LIN {X 0,Y 187.073,Z 696.63,A -85,B 0,C 180,E1 -22033.993,E2 -22033.993} C_VEL
LIN {X 0,Y 186.264,Z 706.069,A -85,B 0,C 180,E1 -22036.36,E2 -22036.36} C_VEL
LIN {X 0,Y 185.581,Z 714.682,A -85,B 0,C 180,E1 -22039.085,E2 -22039.085} C_VEL
LIN {X 0,Y 185.452,Z 722.782,A -85,B 0,C 180,E1 -22042.378,E2 -22042.378} C_VEL
LIN {X 0,Y 185.879,Z 728.927,A -85,B 0,C 180,E1 -22045.663,E2 -22045.663} C_VEL
LIN {X 0,Y 186.509,Z 733.408,A -85,B 0,C 180,E1 -22048.92,E2 -22048.92} C_VEL
LIN {X 0,Y 186.681,Z 734.524,A -85,B 0,C 180,E1 -22050,E2 -22050} C_VEL
LIN {X 0,Y 185.88,Z 736.061,A -85,B 0,C 180,E1 -22052.167,E2 -22052.167} C_VEL
LIN {X 0,Y 185.102,Z 737.03,A -85,B 0,C 180,E1 -22054.355,E2 -22054.355} C_VEL
LIN {X 0,Y 184.441,Z 737.622,A -85,B 0,C 180,E1 -22057.819,E2 -22057.819} C_VEL
LIN {X 0,Y 184.416,Z 737.19,A -85,B 0,C 180,E1 -22060.984,E2 -22060.984} C_VEL
LIN {X 0,Y 184.832,Z 736.376,A -85,B 0,C 180,E1 -22063.187,E2 -22063.187} C_VEL
LIN {X 0,Y 185.593,Z 735.101,A -85,B 0,C 180,E1 -22065.371,E2 -22065.371} C_VEL
LIN {X 0,Y 187.611,Z 732.415,A -85,B 0,C 180,E1 -22068.566,E2 -22068.566} C_VEL
LIN {X 0,Y 190.356,Z 728.663,A -85,B 0,C 180,E1 -22071.666,E2 -22071.666} C_VEL
LIN {X 0,Y 193.883,Z 723.809,A -85,B 0,C 180,E1 -22074.636,E2 -22074.636} C_VEL
LIN {X 0,Y 198.128,Z 717.663,A -85,B 0,C 180,E1 -22077.46,E2 -22077.46} C_VEL
LIN {X 0,Y 203.13,Z 709.985,A -85,B 0,C 180,E1 -22080.11,E2 -22080.11} C_VEL
LIN {X 0,Y 208.674,Z 700.543,A -85,B 0,C 180,E1 -22082.606,E2 -22082.606} C_VEL
LIN {X 0,Y 213.814,Z 690.855,A -85,B 0,C 180,E1 -22084.54,E2 -22084.54} C_VEL
LIN {X 0,Y 218.839,Z 680.033,A -85,B 0,C 180,E1 -22086.164,E2 -22086.164} C_VEL
LIN {X 0,Y 223.644,Z 667.781,A -85,B 0,C 180,E1 -22087.568,E2 -22087.568} C_VEL
LIN {X 0,Y 227.072,Z 655.896,A -85,B 0,C 180,E1 -22088.76,E2 -22088.76} C_VEL
LIN {X 0,Y 229.32,Z 643.699,A -85,B 0,C 180,E1 -22089.904,E2 -22089.904} C_VEL
LIN {X 0,Y 230.194,Z 631.94,A -85,B 0,C 180,E1 -22091.105,E2 -22091.105} C_VEL
LIN {X 0,Y 230.347,Z 618.408,A -85,B 0,C 180,E1 -22092.713,E2 -22092.713} C_VEL
LIN {X 0,Y 230.219,Z 613.273,A -85,B 0,C 180,E1 -22093.463,E2 -22093.463} C_VEL
LIN {X 0,Y 228.941,Z 606.861,A -85,B 0,C 180,E1 -22095.34,E2 -22095.34} C_VEL
LIN {X 0,Y 227.692,Z 600.839,A -85,B 0,C 180,E1 -22097.501,E2 -22097.501} C_VEL
LIN {X 0,Y 227.171,Z 599.159,A -85,B 0,C 180,E1 -22098.473,E2 -22098.473} C_VEL
LIN {X 0,Y 225.431,Z 596.58,A -85,B 0,C 180,E1 -22101.958,E2 -22101.958} C_VEL
LIN {X 0,Y 225.098,Z 595.189,A -85,B 0,C 180,E1 -22103.615,E2 -22103.615} C_VEL
LIN {X 0,Y 224.948,Z 594.902,A -85,B 0,C 180,E1 -22105.781,E2 -22105.781} C_VEL
LIN {X 0,Y 225.214,Z 595.291,A -85,B 0,C 180,E1 -22107.961,E2 -22107.961} C_VEL
LIN {X 0,Y 226.659,Z 598.492,A -85,B 0,C 180,E1 -22111.962,E2 -22111.962} C_VEL
LIN {X 0,Y 227.457,Z 599.455,A -85,B 0,C 180,E1 -22113.163,E2 -22113.163} C_VEL
LIN {X 0,Y 229.844,Z 603.626,A -85,B 0,C 180,E1 -22116.036,E2 -22116.036} C_VEL
LIN {X 0,Y 232.174,Z 607.948,A -85,B 0,C 180,E1 -22118.251,E2 -22118.251} C_VEL
LIN {X 0,Y 234.9,Z 614.48,A -85,B 0,C 180,E1 -22120.836,E2 -22120.836} C_VEL
LIN {X 0,Y 235.052,Z 614.986,A -85,B 0,C 180,E1 -22121,E2 -22121} C_VEL
LIN {X 0,Y 232.571,Z 626.818,A -85,B 0,C 180,E1 -22122.138,E2 -22122.138} C_VEL
LIN {X 0,Y 229.272,Z 638.439,A -85,B 0,C 180,E1 -22123.564,E2 -22123.564} C_VEL
LIN {X 0,Y 225.173,Z 649.567,A -85,B 0,C 180,E1 -22125.36,E2 -22125.36} C_VEL
LIN {X 0,Y 221.221,Z 658.24,A -85,B 0,C 180,E1 -22127.152,E2 -22127.152} C_VEL
LIN {X 0,Y 216.836,Z 666.323,A -85,B 0,C 180,E1 -22129.26,E2 -22129.26} C_VEL
LIN {X 0,Y 212.196,Z 673.689,A -85,B 0,C 180,E1 -22131.705,E2 -22131.705} C_VEL
LIN {X 0,Y 207.957,Z 679.351,A -85,B 0,C 180,E1 -22134.182,E2 -22134.182} C_VEL
LIN {X 0,Y 204.161,Z 683.648,A -85,B 0,C 180,E1 -22136.624,E2 -22136.624} C_VEL
LIN {X 0,Y 199.63,Z 687.906,A -85,B 0,C 180,E1 -22140.001,E2 -22140.001} C_VEL
LIN {X 0,Y 196.952,Z 689.883,A -85,B 0,C 180,E1 -22142.402,E2 -22142.402} C_VEL
LIN {X 0,Y 195.179,Z 690.897,A -85,B 0,C 180,E1 -22144.131,E2 -22144.131} C_VEL
LIN {X 0,Y 193.199,Z 691.679,A -85,B 0,C 180,E1 -22146.266,E2 -22146.266} C_VEL
LIN {X 0,Y 191.455,Z 691.968,A -85,B 0,C 180,E1 -22148.444,E2 -22148.444} C_VEL
LIN {X 0,Y 189.965,Z 691.804,A -85,B 0,C 180,E1 -22150.661,E2 -22150.661} C_VEL
LIN {X 0,Y 188.205,Z 690.717,A -85,B 0,C 180,E1 -22153.863,E2 -22153.863} C_VEL
LIN {X 0,Y 186.809,Z 688.3,A -85,B 0,C 180,E1 -22157.517,E2 -22157.517} C_VEL
LIN {X 0,Y 186.045,Z 684.811,A -85,B 0,C 180,E1 -22161.032,E2 -22161.032} C_VEL
LIN {X 0,Y 185.795,Z 679.7,A -85,B 0,C 180,E1 -22164.795,E2 -22164.795} C_VEL
LIN {X 0,Y 186.113,Z 673.685,A -85,B 0,C 180,E1 -22168.167,E2 -22168.167} C_VEL
LIN {X 0,Y 186.657,Z 666.806,A -85,B 0,C 180,E1 -22171.257,E2 -22171.257} C_VEL
LIN {X 0,Y 187.547,Z 658.71,A -85,B 0,C 180,E1 -22174.202,E2 -22174.202} C_VEL
LIN {X 0,Y 188.726,Z 648.29,A -85,B 0,C 180,E1 -22177.24,E2 -22177.24} C_VEL
LIN {X 0,Y 189.888,Z 637.77,A -85,B 0,C 180,E1 -22179.677,E2 -22179.677} C_VEL
LIN {X 0,Y 191.08,Z 626.638,A -85,B 0,C 180,E1 -22181.739,E2 -22181.739} C_VEL
LIN {X 0,Y 192.124,Z 614.599,A -85,B 0,C 180,E1 -22183.476,E2 -22183.476} C_VEL
LIN {X 0,Y 193.024,Z 600.995,A -85,B 0,C 180,E1 -22184.933,E2 -22184.933} C_VEL
LIN {X 0,Y 193.538,Z 586.899,A -85,B 0,C 180,E1 -22185.94,E2 -22185.94} C_VEL
LIN {X 0,Y 193.468,Z 578.507,A -85,B 0,C 180,E1 -22186.408,E2 -22186.408} C_VEL
LIN {X 0,Y 185.856,Z 553.298,A -85,B 0,C 180,E1 -22188.311,E2 -22188.311} C_VEL
LIN {X 0,Y 185.644,Z 552.294,A -85,B 0,C 180,E1 -22188.703,E2 -22188.703} C_VEL
LIN {X 0,Y 185.561,Z 552.183,A -85,B 0,C 180,E1 -22192.701,E2 -22192.701} C_VEL
LIN {X 0,Y 185.547,Z 552.185,A -85,B 0,C 180,E1 -22197.977,E2 -22197.977} C_VEL
LIN {X 0,Y 185.584,Z 552.179,A -85,B 0,C 180,E1 -22200.577,E2 -22200.577} C_VEL
LIN {X 0,Y 185.591,Z 552.18,A -85,B 0,C 180,E1 -22205.384,E2 -22205.384} C_VEL
LIN {X 0,Y 185.676,Z 552.168,A -85,B 0,C 180,E1 -22211.136,E2 -22211.136} C_VEL
LIN {X 0,Y 185.686,Z 552.163,A -85,B 0,C 180,E1 -22214.637,E2 -22214.637} C_VEL
LIN {X 0,Y 185.892,Z 552.142,A -85,B 0,C 180,E1 -22219.419,E2 -22219.419} C_VEL
LIN {X 0,Y 185.945,Z 552.131,A -85,B 0,C 180,E1 -22223.49,E2 -22223.49} C_VEL
LIN {X 0,Y 186.209,Z 552.103,A -85,B 0,C 180,E1 -22227.837,E2 -22227.837} C_VEL
LIN {X 0,Y 186.411,Z 552.074,A -85,B 0,C 180,E1 -22230,E2 -22230} C_VEL
LIN {X 0,Y 185.918,Z 552.138,A -85,B 0,C 180,E1 -22234.336,E2 -22234.336} C_VEL
LIN {X 0,Y 185.983,Z 552.127,A -85,B 0,C 180,E1 -22238.694,E2 -22238.694} C_VEL
LIN {X 0,Y 185.734,Z 552.159,A -85,B 0,C 180,E1 -22243.122,E2 -22243.122} C_VEL
LIN {X 0,Y 185.694,Z 552.166,A -85,B 0,C 180,E1 -22247.624,E2 -22247.624} C_VEL
LIN {X 0,Y 185.585,Z 552.18,A -85,B 0,C 180,E1 -22252.252,E2 -22252.252} C_VEL
LIN {X 0,Y 185.561,Z 552.178,A -85,B 0,C 180,E1 -22257.032,E2 -22257.032} C_VEL
LIN {X 0,Y 185.58,Z 552.177,A -85,B 0,C 180,E1 -22259.492,E2 -22259.492} C_VEL
LIN {X 0,Y 185.522,Z 552.185,A -85,B 0,C 180,E1 -22264.626,E2 -22264.626} C_VEL
LIN {X 0,Y 185.57,Z 552.175,A -85,B 0,C 180,E1 -22267.313,E2 -22267.313} C_VEL
LIN {X 0,Y 185.563,Z 552.182,A -85,B 0,C 180,E1 -22270.756,E2 -22270.756} C_VEL
LIN {X 0,Y 185.555,Z 552.183,A -85,B 0,C 180,E1 -22273.974,E2 -22273.974} C_VEL
LIN {X 0,Y 185.493,Z 552.19,A -85,B 0,C 180,E1 -22279.266,E2 -22279.266} C_VEL
LIN {X 0,Y 185.544,Z 552.182,A -85,B 0,C 180,E1 -22282.695,E2 -22282.695} C_VEL
LIN {X 0,Y 185.544,Z 552.185,A -85,B 0,C 180,E1 -22287.974,E2 -22287.974} C_VEL
LIN {X 0,Y 185.581,Z 552.18,A -85,B 0,C 180,E1 -22290.575,E2 -22290.575} C_VEL
LIN {X 0,Y 185.605,Z 552.174,A -85,B 0,C 180,E1 -22295.384,E2 -22295.384} C_VEL
LIN {X 0,Y 185.708,Z 552.161,A -85,B 0,C 180,E1 -22301.101,E2 -22301.101} C_VEL
LIN {X 0,Y 185.731,Z 552.161,A -85,B 0,C 180,E1 -22306.876,E2 -22306.876} C_VEL
LIN {X 0,Y 186.011,Z 552.12,A -85,B 0,C 180,E1 -22311.307,E2 -22311.307} C_VEL
LIN {X 0,Y 186.205,Z 552.101,A -85,B 0,C 180,E1 -22317.836,E2 -22317.836} C_VEL
LIN {X 0,Y 186.403,Z 552.074,A -85,B 0,C 180,E1 -22319.999,E2 -22319.999} C_VEL
LIN {X 0,Y 185.92,Z 552.139,A -85,B 0,C 180,E1 -22324.335,E2 -22324.335} C_VEL
LIN {X 0,Y 186.005,Z 552.124,A -85,B 0,C 180,E1 -22328.692,E2 -22328.692} C_VEL
LIN {X 0,Y 185.76,Z 552.158,A -85,B 0,C 180,E1 -22333.12,E2 -22333.12} C_VEL
LIN {X 0,Y 185.67,Z 552.167,A -85,B 0,C 180,E1 -22338.865,E2 -22338.865} C_VEL
LIN {X 0,Y 185.574,Z 552.181,A -85,B 0,C 180,E1 -22344.646,E2 -22344.646} C_VEL
LIN {X 0,Y 185.576,Z 552.179,A -85,B 0,C 180,E1 -22349.493,E2 -22349.493} C_VEL
LIN {X 0,Y 185.496,Z 552.189,A -85,B 0,C 180,E1 -22354.632,E2 -22354.632} C_VEL
LIN {X 0,Y 185.502,Z 552.188,A -85,B 0,C 180,E1 -22357.313,E2 -22357.313} C_VEL
LIN {X 0,Y 185.468,Z 552.196,A -85,B 0,C 180,E1 -22360.725,E2 -22360.725} C_VEL
LIN {X 0,Y 185.481,Z 552.192,A -85,B 0,C 180,E1 -22366.047,E2 -22366.047} C_VEL
LIN {X 0,Y 185.546,Z 552.184,A -85,B 0,C 180,E1 -22369.917,E2 -22369.917} C_VEL
LIN {X 0,Y 185.936,Z 552.249,A -85,B 0,C 180,E1 -22373.802,E2 -22373.802} C_VEL
LIN {X 0,Y 188.152,Z 562.25,A -85,B 0,C 180,E1 -22379.216,E2 -22379.216} C_VEL
LIN {X 0,Y 187.814,Z 565.476,A -85,B 0,C 180,E1 -22380.892,E2 -22380.892} C_VEL
LIN {X 0,Y 187.128,Z 569.009,A -85,B 0,C 180,E1 -22382.609,E2 -22382.609} C_VEL
LIN {X 0,Y 187.031,Z 577.205,A -85,B 0,C 180,E1 -22383.198,E2 -22383.198} C_VEL
LIN {X 0,Y 188.442,Z 619.399,A -85,B 0,C 180,E1 -22385.888,E2 -22385.888} C_VEL
LIN {X 0,Y 190.503,Z 655.952,A -85,B 0,C 180,E1 -22388.293,E2 -22388.293} C_VEL
LIN {X 0,Y 189.725,Z 669.284,A -85,B 0,C 180,E1 -22389.538,E2 -22389.538} C_VEL
LIN {X 0,Y 188.888,Z 680.435,A -85,B 0,C 180,E1 -22391.001,E2 -22391.001} C_VEL
LIN {X 0,Y 187.691,Z 691.166,A -85,B 0,C 180,E1 -22392.85,E2 -22392.85} C_VEL
LIN {X 0,Y 187.073,Z 696.63,A -85,B 0,C 180,E1 -22393.993,E2 -22393.993} C_VEL
LIN {X 0,Y 186.033,Z 701.223,A -85,B 0,C 180,E1 -22395.088,E2 -22395.088} C_VEL
LIN {X 0,Y 184.084,Z 705.387,A -85,B 0,C 180,E1 -22396.259,E2 -22396.259} C_VEL
LIN {X 0,Y 179.28,Z 714.053,A -85,B 0,C 180,E1 -22399.363,E2 -22399.363} C_VEL
LIN {X 0,Y 178.5,Z 717.649,A -85,B 0,C 180,E1 -22400.862,E2 -22400.862} C_VEL
LIN {X 0,Y 178.611,Z 723.876,A -85,B 0,C 180,E1 -22403.788,E2 -22403.788} C_VEL
LIN {X 0,Y 179.114,Z 728.664,A -85,B 0,C 180,E1 -22406.626,E2 -22406.626} C_VEL
LIN {X 0,Y 179.742,Z 732.818,A -85,B 0,C 180,E1 -22410,E2 -22410} C_VEL
LIN {X 0,Y 178.911,Z 734.455,A -85,B 0,C 180,E1 -22412.251,E2 -22412.251} C_VEL
LIN {X 0,Y 178.117,Z 735.55,A -85,B 0,C 180,E1 -22414.526,E2 -22414.526} C_VEL
LIN {X 0,Y 177.451,Z 736.328,A -85,B 0,C 180,E1 -22418.061,E2 -22418.061} C_VEL
LIN {X 0,Y 177.457,Z 736.091,A -85,B 0,C 180,E1 -22421.421,E2 -22421.421} C_VEL
LIN {X 0,Y 177.911,Z 735.399,A -85,B 0,C 180,E1 -22423.71,E2 -22423.71} C_VEL
LIN {X 0,Y 178.744,Z 734.306,A -85,B 0,C 180,E1 -22425.975,E2 -22425.975} C_VEL
LIN {X 0,Y 180.087,Z 732.766,A -85,B 0,C 180,E1 -22428.192,E2 -22428.192} C_VEL
LIN {X 0,Y 182.694,Z 729.638,A -85,B 0,C 180,E1 -22431.435,E2 -22431.435} C_VEL
LIN {X 0,Y 186.137,Z 725.46,A -85,B 0,C 180,E1 -22434.539,E2 -22434.539} C_VEL
LIN {X 0,Y 190.307,Z 720.092,A -85,B 0,C 180,E1 -22437.491,E2 -22437.491} C_VEL
LIN {X 0,Y 195.237,Z 713.418,A -85,B 0,C 180,E1 -22440.261,E2 -22440.261} C_VEL
LIN {X 0,Y 200.824,Z 705.139,A -85,B 0,C 180,E1 -22442.848,E2 -22442.848} C_VEL
LIN {X 0,Y 205.901,Z 696.719,A -85,B 0,C 180,E1 -22444.87,E2 -22444.87} C_VEL
LIN {X 0,Y 211.445,Z 686.511,A -85,B 0,C 180,E1 -22446.746,E2 -22446.746} C_VEL
LIN {X 0,Y 216.807,Z 675.161,A -85,B 0,C 180,E1 -22448.311,E2 -22448.311} C_VEL
LIN {X 0,Y 221.508,Z 662.765,A -85,B 0,C 180,E1 -22449.655,E2 -22449.655} C_VEL
LIN {X 0,Y 225.007,Z 649.325,A -85,B 0,C 180,E1 -22450.989,E2 -22450.989} C_VEL
LIN {X 0,Y 226.845,Z 637.084,A -85,B 0,C 180,E1 -22452.264,E2 -22452.264} C_VEL
LIN {X 0,Y 227.432,Z 624.858,A -85,B 0,C 180,E1 -22453.702,E2 -22453.702} C_VEL
LIN {X 0,Y 227.525,Z 617.57,A -85,B 0,C 180,E1 -22454.73,E2 -22454.73} C_VEL
LIN {X 0,Y 226.586,Z 612.063,A -85,B 0,C 180,E1 -22456.419,E2 -22456.419} C_VEL
LIN {X 0,Y 225.732,Z 606.668,A -85,B 0,C 180,E1 -22458.405,E2 -22458.405} C_VEL
LIN {X 0,Y 225.345,Z 605.805,A -85,B 0,C 180,E1 -22459.086,E2 -22459.086} C_VEL
LIN {X 0,Y 223.72,Z 602.433,A -85,B 0,C 180,E1 -22463.455,E2 -22463.455} C_VEL
LIN {X 0,Y 223.648,Z 601.921,A -85,B 0,C 180,E1 -22464.787,E2 -22464.787} C_VEL
LIN {X 0,Y 223.817,Z 602.217,A -85,B 0,C 180,E1 -22467.737,E2 -22467.737} C_VEL
LIN {X 0,Y 225.184,Z 605.393,A -85,B 0,C 180,E1 -22471.762,E2 -22471.762} C_VEL
LIN {X 0,Y 225.852,Z 606.361,A -85,B 0,C 180,E1 -22472.877,E2 -22472.877} C_VEL
LIN {X 0,Y 227.992,Z 610.487,A -85,B 0,C 180,E1 -22475.714,E2 -22475.714} C_VEL
LIN {X 0,Y 229.929,Z 614.71,A -85,B 0,C 180,E1 -22477.925,E2 -22477.925} C_VEL
LIN {X 0,Y 231.347,Z 619.083,A -85,B 0,C 180,E1 -22479.72,E2 -22479.72} C_VEL
LIN {X 0,Y 228.581,Z 630.79,A -85,B 0,C 180,E1 -22480.905,E2 -22480.905} C_VEL
LIN {X 0,Y 225.152,Z 641.388,A -85,B 0,C 180,E1 -22482.282,E2 -22482.282} C_VEL
LIN {X 0,Y 221.407,Z 650.703,A -85,B 0,C 180,E1 -22483.815,E2 -22483.815} C_VEL
LIN {X 0,Y 217.257,Z 659.441,A -85,B 0,C 180,E1 -22485.613,E2 -22485.613} C_VEL
LIN {X 0,Y 212.83,Z 667.182,A -85,B 0,C 180,E1 -22487.606,E2 -22487.606} C_VEL
LIN {X 0,Y 207.533,Z 675.048,A -85,B 0,C 180,E1 -22490.252,E2 -22490.252} C_VEL
LIN {X 0,Y 202.496,Z 681.229,A -85,B 0,C 180,E1 -22493.024,E2 -22493.024} C_VEL
LIN {X 0,Y 197.859,Z 686.015,A -85,B 0,C 180,E1 -22495.927,E2 -22495.927} C_VEL
LIN {X 0,Y 195.01,Z 688.451,A -85,B 0,C 180,E1 -22497.935,E2 -22497.935} C_VEL
LIN {X 0,Y 192.388,Z 690.37,A -85,B 0,C 180,E1 -22500.001,E2 -22500.001} C_VEL
LIN {X 0,Y 189.895,Z 691.813,A -85,B 0,C 180,E1 -22502.229,E2 -22502.229} C_VEL
LIN {X 0,Y 187.822,Z 692.692,A -85,B 0,C 180,E1 -22504.293,E2 -22504.293} C_VEL
LIN {X 0,Y 184.566,Z 693.194,A -85,B 0,C 180,E1 -22508.105,E2 -22508.105} C_VEL
LIN {X 0,Y 182.57,Z 692.633,A -85,B 0,C 180,E1 -22511.098,E2 -22511.098} C_VEL
LIN {X 0,Y 181.043,Z 691.349,A -85,B 0,C 180,E1 -22513.961,E2 -22513.961} C_VEL
LIN {X 0,Y 179.879,Z 689.194,A -85,B 0,C 180,E1 -22517.04,E2 -22517.04} C_VEL
LIN {X 0,Y 179.007,Z 685.579,A -85,B 0,C 180,E1 -22520.693,E2 -22520.693} C_VEL
LIN {X 0,Y 178.724,Z 680.904,A -85,B 0,C 180,E1 -22524.205,E2 -22524.205} C_VEL
LIN {X 0,Y 178.998,Z 674.136,A -85,B 0,C 180,E1 -22528.11,E2 -22528.11} C_VEL
LIN {X 0,Y 179.537,Z 667.323,A -85,B 0,C 180,E1 -22531.244,E2 -22531.244} C_VEL
LIN {X 0,Y 180.491,Z 658.88,A -85,B 0,C 180,E1 -22534.376,E2 -22534.376} C_VEL
LIN {X 0,Y 181.534,Z 649.389,A -85,B 0,C 180,E1 -22537.224,E2 -22537.224} C_VEL
LIN {X 0,Y 182.757,Z 638.966,A -85,B 0,C 180,E1 -22539.728,E2 -22539.728} C_VEL
LIN {X 0,Y 183.988,Z 627.382,A -85,B 0,C 180,E1 -22541.95,E2 -22541.95} C_VEL
LIN {X 0,Y 185.129,Z 614.5,A -85,B 0,C 180,E1 -22543.84,E2 -22543.84} C_VEL
LIN {X 0,Y 185.988,Z 602.146,A -85,B 0,C 180,E1 -22545.191,E2 -22545.191} C_VEL
LIN {X 0,Y 186.568,Z 587.713,A -85,B 0,C 180,E1 -22546.257,E2 -22546.257} C_VEL
LIN {X 0,Y 186.617,Z 580.167,A -85,B 0,C 180,E1 -22546.69,E2 -22546.69} C_VEL
LIN {X 0,Y 178.719,Z 553.941,A -85,B 0,C 180,E1 -22548.778,E2 -22548.778} C_VEL
LIN {X 0,Y 178.543,Z 553.135,A -85,B 0,C 180,E1 -22549.203,E2 -22549.203} C_VEL
LIN {X 0,Y 178.46,Z 553.068,A -85,B 0,C 180,E1 -22553.793,E2 -22553.793} C_VEL
LIN {X 0,Y 178.493,Z 553.063,A -85,B 0,C 180,E1 -22556.549,E2 -22556.549} C_VEL
LIN {X 0,Y 178.525,Z 553.059,A -85,B 0,C 180,E1 -22560.007,E2 -22560.007} C_VEL
LIN {X 0,Y 178.537,Z 553.057,A -85,B 0,C 180,E1 -22564.877,E2 -22564.877} C_VEL
LIN {X 0,Y 178.624,Z 553.045,A -85,B 0,C 180,E1 -22570.787,E2 -22570.787} C_VEL
LIN {X 0,Y 178.654,Z 553.042,A -85,B 0,C 180,E1 -22576.348,E2 -22576.348} C_VEL
LIN {X 0,Y 178.912,Z 553.008,A -85,B 0,C 180,E1 -22580.96,E2 -22580.96} C_VEL
LIN {X 0,Y 179.154,Z 552.982,A -85,B 0,C 180,E1 -22587.752,E2 -22587.752} C_VEL
LIN {X 0,Y 179.374,Z 552.95,A -85,B 0,C 180,E1 -22590,E2 -22590} C_VEL
LIN {X 0,Y 178.866,Z 553.016,A -85,B 0,C 180,E1 -22594.507,E2 -22594.507} C_VEL
LIN {X 0,Y 178.912,Z 553.007,A -85,B 0,C 180,E1 -22599.04,E2 -22599.04} C_VEL
LIN {X 0,Y 178.662,Z 553.042,A -85,B 0,C 180,E1 -22603.652,E2 -22603.652} C_VEL
LIN {X 0,Y 178.626,Z 553.041,A -85,B 0,C 180,E1 -22609.215,E2 -22609.215} C_VEL
LIN {X 0,Y 178.523,Z 553.058,A -85,B 0,C 180,E1 -22615.113,E2 -22615.113} C_VEL
LIN {X 0,Y 178.524,Z 553.058,A -85,B 0,C 180,E1 -22619.992,E2 -22619.992} C_VEL
LIN {X 0,Y 178.486,Z 553.063,A -85,B 0,C 180,E1 -22624.218,E2 -22624.218} C_VEL
LIN {X 0,Y 178.474,Z 553.063,A -85,B 0,C 180,E1 -22629.053,E2 -22629.053} C_VEL
LIN {X 0,Y 178.499,Z 553.064,A -85,B 0,C 180,E1 -22632.015,E2 -22632.015} C_VEL
LIN {X 0,Y 178.457,Z 553.063,A -85,B 0,C 180,E1 -22635.143,E2 -22635.143} C_VEL
LIN {X 0,Y 178.424,Z 553.072,A -85,B 0,C 180,E1 -22638.45,E2 -22638.45} C_VEL
LIN {X 0,Y 178.449,Z 553.066,A -85,B 0,C 180,E1 -22643.788,E2 -22643.788} C_VEL
LIN {X 0,Y 178.49,Z 553.063,A -85,B 0,C 180,E1 -22646.546,E2 -22646.546} C_VEL
LIN {X 0,Y 178.522,Z 553.061,A -85,B 0,C 180,E1 -22650.005,E2 -22650.005} C_VEL
LIN {X 0,Y 178.534,Z 553.055,A -85,B 0,C 180,E1 -22654.874,E2 -22654.874} C_VEL
LIN {X 0,Y 178.651,Z 553.04,A -85,B 0,C 180,E1 -22660.755,E2 -22660.755} C_VEL
LIN {X 0,Y 178.659,Z 553.044,A -85,B 0,C 180,E1 -22666.347,E2 -22666.347} C_VEL
LIN {X 0,Y 178.961,Z 552.999,A -85,B 0,C 180,E1 -22670.961,E2 -22670.961} C_VEL
LIN {X 0,Y 179.151,Z 552.98,A -85,B 0,C 180,E1 -22677.751,E2 -22677.751} C_VEL
LIN {X 0,Y 179.366,Z 552.951,A -85,B 0,C 180,E1 -22679.999,E2 -22679.999} C_VEL
LIN {X 0,Y 178.869,Z 553.018,A -85,B 0,C 180,E1 -22684.506,E2 -22684.506} C_VEL
LIN {X 0,Y 178.934,Z 553.003,A -85,B 0,C 180,E1 -22689.038,E2 -22689.038} C_VEL
LIN {X 0,Y 178.677,Z 553.039,A -85,B 0,C 180,E1 -22693.65,E2 -22693.65} C_VEL
LIN {X 0,Y 178.617,Z 553.045,A -85,B 0,C 180,E1 -22699.213,E2 -22699.213} C_VEL
LIN {X 0,Y 178.516,Z 553.058,A -85,B 0,C 180,E1 -22705.114,E2 -22705.114} C_VEL
LIN {X 0,Y 178.498,Z 553.064,A -85,B 0,C 180,E1 -22710.786,E2 -22710.786} C_VEL
LIN {X 0,Y 178.482,Z 553.063,A -85,B 0,C 180,E1 -22714.219,E2 -22714.219} C_VEL
LIN {X 0,Y 178.392,Z 553.076,A -85,B 0,C 180,E1 -22719.074,E2 -22719.074} C_VEL
LIN {X 0,Y 178.396,Z 553.074,A -85,B 0,C 180,E1 -22722.045,E2 -22722.045} C_VEL
LIN {X 0,Y 178.401,Z 553.075,A -85,B 0,C 180,E1 -22725.161,E2 -22725.161} C_VEL
LIN {X 0,Y 178.532,Z 553.06,A -85,B 0,C 180,E1 -22730.962,E2 -22730.962} C_VEL
LIN {X 0,Y 178.947,Z 553.155,A -85,B 0,C 180,E1 -22734.096,E2 -22734.096} C_VEL
LIN {X 0,Y 180.808,Z 561.446,A -85,B 0,C 180,E1 -22738.774,E2 -22738.774} C_VEL
LIN {X 0,Y 180.938,Z 564.291,A -85,B 0,C 180,E1 -22740.315,E2 -22740.315} C_VEL
LIN {X 0,Y 180.257,Z 567.596,A -85,B 0,C 180,E1 -22742.026,E2 -22742.026} C_VEL
LIN {X 0,Y 180.117,Z 573.051,A -85,B 0,C 180,E1 -22742.48,E2 -22742.48} C_VEL
LIN {X 0,Y 180.81,Z 605.623,A -85,B 0,C 180,E1 -22744.652,E2 -22744.652} C_VEL
LIN {X 0,Y 183.445,Z 655.478,A -85,B 0,C 180,E1 -22748.067,E2 -22748.067} C_VEL
LIN {X 0,Y 182.729,Z 668.104,A -85,B 0,C 180,E1 -22749.307,E2 -22749.307} C_VEL
LIN {X 0,Y 181.897,Z 679.224,A -85,B 0,C 180,E1 -22750.828,E2 -22750.828} C_VEL
LIN {X 0,Y 180.706,Z 689.958,A -85,B 0,C 180,E1 -22752.75,E2 -22752.75} C_VEL
LIN {X 0,Y 179.625,Z 699.71,A -85,B 0,C 180,E1 -22754.977,E2 -22754.977} C_VEL
LIN {X 0,Y 178.966,Z 708.573,A -85,B 0,C 180,E1 -22757.527,E2 -22757.527} C_VEL
LIN {X 0,Y 178.513,Z 716.871,A -85,B 0,C 180,E1 -22760.532,E2 -22760.532} C_VEL
LIN {X 0,Y 178.5,Z 717.649,A -85,B 0,C 180,E1 -22760.862,E2 -22760.862} C_VEL
LIN {X 0,Y 178.053,Z 721.046,A -85,B 0,C 180,E1 -22762.422,E2 -22762.422} C_VEL
LIN {X 0,Y 177.018,Z 724.021,A -85,B 0,C 180,E1 -22764.053,E2 -22764.053} C_VEL
LIN {X 0,Y 176.142,Z 725.771,A -85,B 0,C 180,E1 -22765.176,E2 -22765.176} C_VEL
LIN {X 0,Y 173.45,Z 729.979,A -85,B 0,C 180,E1 -22768.766,E2 -22768.766} C_VEL
LIN {X 0,Y 172.796,Z 731.035,A -85,B 0,C 180,E1 -22770.029,E2 -22770.029} C_VEL
LIN {X 0,Y 171.96,Z 732.784,A -85,B 0,C 180,E1 -22772.342,E2 -22772.342} C_VEL
LIN {X 0,Y 171.16,Z 734.013,A -85,B 0,C 180,E1 -22774.71,E2 -22774.71} C_VEL
LIN {X 0,Y 170.456,Z 734.967,A -85,B 0,C 180,E1 -22778.302,E2 -22778.302} C_VEL
LIN {X 0,Y 170.516,Z 734.937,A -85,B 0,C 180,E1 -22781.892,E2 -22781.892} C_VEL
LIN {X 0,Y 171.014,Z 734.404,A -85,B 0,C 180,E1 -22784.274,E2 -22784.274} C_VEL
LIN {X 0,Y 171.924,Z 733.425,A -85,B 0,C 180,E1 -22786.627,E2 -22786.627} C_VEL
LIN {X 0,Y 173.339,Z 732.075,A -85,B 0,C 180,E1 -22788.926,E2 -22788.926} C_VEL
LIN {X 0,Y 176.103,Z 729.219,A -85,B 0,C 180,E1 -22792.279,E2 -22792.279} C_VEL
LIN {X 0,Y 179.696,Z 725.321,A -85,B 0,C 180,E1 -22795.48,E2 -22795.48} C_VEL
LIN {X 0,Y 184.057,Z 720.321,A -85,B 0,C 180,E1 -22798.508,E2 -22798.508} C_VEL
LIN {X 0,Y 190.101,Z 712.857,A -85,B 0,C 180,E1 -22801.79,E2 -22801.79} C_VEL
LIN {X 0,Y 195.944,Z 704.787,A -85,B 0,C 180,E1 -22804.395,E2 -22804.395} C_VEL
LIN {X 0,Y 201.286,Z 696.68,A -85,B 0,C 180,E1 -22806.409,E2 -22806.409} C_VEL
LIN {X 0,Y 207.059,Z 686.823,A -85,B 0,C 180,E1 -22808.274,E2 -22808.274} C_VEL
LIN {X 0,Y 212.619,Z 675.863,A -85,B 0,C 180,E1 -22809.822,E2 -22809.822} C_VEL
LIN {X 0,Y 217.396,Z 664.559,A -85,B 0,C 180,E1 -22811.098,E2 -22811.098} C_VEL
LIN {X 0,Y 221.11,Z 652.568,A -85,B 0,C 180,E1 -22812.356,E2 -22812.356} C_VEL
LIN {X 0,Y 223.367,Z 641.345,A -85,B 0,C 180,E1 -22813.563,E2 -22813.563} C_VEL
LIN {X 0,Y 224.702,Z 629.481,A -85,B 0,C 180,E1 -22814.982,E2 -22814.982} C_VEL
LIN {X 0,Y 225.026,Z 621.981,A -85,B 0,C 180,E1 -22816.028,E2 -22816.028} C_VEL
LIN {X 0,Y 224.389,Z 617.43,A -85,B 0,C 180,E1 -22817.479,E2 -22817.479} C_VEL
LIN {X 0,Y 223.884,Z 612.811,A -85,B 0,C 180,E1 -22819.173,E2 -22819.173} C_VEL
LIN {X 0,Y 222.33,Z 608.988,A -85,B 0,C 180,E1 -22824.268,E2 -22824.268} C_VEL
LIN {X 0,Y 222.409,Z 609.045,A -85,B 0,C 180,E1 -22827.381,E2 -22827.381} C_VEL
LIN {X 0,Y 224.124,Z 613.06,A -85,B 0,C 180,E1 -22832.423,E2 -22832.423} C_VEL
LIN {X 0,Y 225.755,Z 616.789,A -85,B 0,C 180,E1 -22835.114,E2 -22835.114} C_VEL
LIN {X 0,Y 227.076,Z 620.391,A -85,B 0,C 180,E1 -22837.129,E2 -22837.129} C_VEL
LIN {X 0,Y 227.737,Z 622.939,A -85,B 0,C 180,E1 -22838.265,E2 -22838.265} C_VEL
LIN {X 0,Y 227.65,Z 623.959,A -85,B 0,C 180,E1 -22838.47,E2 -22838.47} C_VEL
LIN {X 0,Y 224.16,Z 636.213,A -85,B 0,C 180,E1 -22839.826,E2 -22839.826} C_VEL
LIN {X 0,Y 220.592,Z 645.925,A -85,B 0,C 180,E1 -22841.182,E2 -22841.182} C_VEL
LIN {X 0,Y 216.027,Z 655.965,A -85,B 0,C 180,E1 -22842.975,E2 -22842.975} C_VEL
LIN {X 0,Y 210.933,Z 665.059,A -85,B 0,C 180,E1 -22845.065,E2 -22845.065} C_VEL
LIN {X 0,Y 205.271,Z 673.58,A -85,B 0,C 180,E1 -22847.645,E2 -22847.645} C_VEL
LIN {X 0,Y 199.528,Z 680.616,A -85,B 0,C 180,E1 -22850.478,E2 -22850.478} C_VEL
LIN {X 0,Y 195.469,Z 684.838,A -85,B 0,C 180,E1 -22852.771,E2 -22852.771} C_VEL
LIN {X 0,Y 190.184,Z 689.391,A -85,B 0,C 180,E1 -22856.132,E2 -22856.132} C_VEL
LIN {X 0,Y 187.786,Z 691.068,A -85,B 0,C 180,E1 -22857.856,E2 -22857.856} C_VEL
LIN {X 0,Y 185.106,Z 692.639,A -85,B 0,C 180,E1 -22860.001,E2 -22860.001} C_VEL
LIN {X 0,Y 182.66,Z 693.702,A -85,B 0,C 180,E1 -22862.206,E2 -22862.206} C_VEL
LIN {X 0,Y 180.415,Z 694.29,A -85,B 0,C 180,E1 -22864.469,E2 -22864.469} C_VEL
LIN {X 0,Y 177.433,Z 694.298,A -85,B 0,C 180,E1 -22868.025,E2 -22868.025} C_VEL
LIN {X 0,Y 175.148,Z 693.233,A -85,B 0,C 180,E1 -22871.575,E2 -22871.575} C_VEL
LIN {X 0,Y 173.879,Z 691.865,A -85,B 0,C 180,E1 -22874.063,E2 -22874.063} C_VEL
LIN {X 0,Y 172.553,Z 688.931,A -85,B 0,C 180,E1 -22877.787,E2 -22877.787} C_VEL
LIN {X 0,Y 171.801,Z 684.767,A -85,B 0,C 180,E1 -22881.604,E2 -22881.604} C_VEL
LIN {X 0,Y 171.661,Z 678.672,A -85,B 0,C 180,E1 -22885.752,E2 -22885.752} C_VEL
LIN {X 0,Y 172.104,Z 671.926,A -85,B 0,C 180,E1 -22889.344,E2 -22889.344} C_VEL
LIN {X 0,Y 172.808,Z 664.298,A -85,B 0,C 180,E1 -22892.608,E2 -22892.608} C_VEL
LIN {X 0,Y 173.762,Z 655.69,A -85,B 0,C 180,E1 -22895.605,E2 -22895.605} C_VEL
LIN {X 0,Y 174.957,Z 645.411,A -85,B 0,C 180,E1 -22898.51,E2 -22898.51} C_VEL
LIN {X 0,Y 176.377,Z 633.29,A -85,B 0,C 180,E1 -22901.203,E2 -22901.203} C_VEL
LIN {X 0,Y 177.535,Z 621.334,A -85,B 0,C 180,E1 -22903.264,E2 -22903.264} C_VEL
LIN {X 0,Y 178.538,Z 608.992,A -85,B 0,C 180,E1 -22904.884,E2 -22904.884} C_VEL
LIN {X 0,Y 179.343,Z 595.321,A -85,B 0,C 180,E1 -22906.144,E2 -22906.144} C_VEL
LIN {X 0,Y 179.631,Z 581.26,A -85,B 0,C 180,E1 -22907.031,E2 -22907.031} C_VEL
LIN {X 0,Y 171.652,Z 554.832,A -85,B 0,C 180,E1 -22909.223,E2 -22909.223} C_VEL
LIN {X 0,Y 171.503,Z 553.996,A -85,B 0,C 180,E1 -22909.698,E2 -22909.698} C_VEL
LIN {X 0,Y 171.409,Z 553.947,A -85,B 0,C 180,E1 -22915.089,E2 -22915.089} C_VEL
LIN {X 0,Y 171.452,Z 553.94,A -85,B 0,C 180,E1 -22920.536,E2 -22920.536} C_VEL
LIN {X 0,Y 171.459,Z 553.938,A -85,B 0,C 180,E1 -22925.803,E2 -22925.803} C_VEL
LIN {X 0,Y 171.58,Z 553.923,A -85,B 0,C 180,E1 -22930.872,E2 -22930.872} C_VEL
LIN {X 0,Y 171.571,Z 553.925,A -85,B 0,C 180,E1 -22935.773,E2 -22935.773} C_VEL
LIN {X 0,Y 171.85,Z 553.888,A -85,B 0,C 180,E1 -22940.585,E2 -22940.585} C_VEL
LIN {X 0,Y 171.813,Z 553.894,A -85,B 0,C 180,E1 -22945.308,E2 -22945.308} C_VEL
LIN {X 0,Y 172.337,Z 553.826,A -85,B 0,C 180,E1 -22950,E2 -22950} C_VEL
LIN {X 0,Y 171.814,Z 553.894,A -85,B 0,C 180,E1 -22954.693,E2 -22954.693} C_VEL
LIN {X 0,Y 171.85,Z 553.888,A -85,B 0,C 180,E1 -22959.415,E2 -22959.415} C_VEL
LIN {X 0,Y 171.58,Z 553.925,A -85,B 0,C 180,E1 -22964.227,E2 -22964.227} C_VEL
LIN {X 0,Y 171.545,Z 553.923,A -85,B 0,C 180,E1 -22969.559,E2 -22969.559} C_VEL
LIN {X 0,Y 171.461,Z 553.939,A -85,B 0,C 180,E1 -22975.608,E2 -22975.608} C_VEL
LIN {X 0,Y 171.442,Z 553.94,A -85,B 0,C 180,E1 -22980.585,E2 -22980.585} C_VEL
LIN {X 0,Y 171.405,Z 553.943,A -85,B 0,C 180,E1 -22985.031,E2 -22985.031} C_VEL
LIN {X 0,Y 171.429,Z 553.941,A -85,B 0,C 180,E1 -22988.835,E2 -22988.835} C_VEL
LIN {X 0,Y 171.387,Z 553.946,A -85,B 0,C 180,E1 -22994.195,E2 -22994.195} C_VEL
LIN {X 0,Y 171.355,Z 553.951,A -85,B 0,C 180,E1 -22998.986,E2 -22998.986} C_VEL
LIN {X 0,Y 171.415,Z 553.946,A -85,B 0,C 180,E1 -23002.047,E2 -23002.047} C_VEL
LIN {X 0,Y 171.41,Z 553.94,A -85,B 0,C 180,E1 -23005.085,E2 -23005.085} C_VEL
LIN {X 0,Y 171.449,Z 553.94,A -85,B 0,C 180,E1 -23010.533,E2 -23010.533} C_VEL
LIN {X 0,Y 171.463,Z 553.936,A -85,B 0,C 180,E1 -23015.801,E2 -23015.801} C_VEL
LIN {X 0,Y 171.607,Z 553.917,A -85,B 0,C 180,E1 -23020.874,E2 -23020.874} C_VEL
LIN {X 0,Y 171.579,Z 553.923,A -85,B 0,C 180,E1 -23025.772,E2 -23025.772} C_VEL
LIN {X 0,Y 171.888,Z 553.881,A -85,B 0,C 180,E1 -23030.586,E2 -23030.586} C_VEL
LIN {X 0,Y 171.82,Z 553.893,A -85,B 0,C 180,E1 -23035.307,E2 -23035.307} C_VEL
LIN {X 0,Y 172.329,Z 553.827,A -85,B 0,C 180,E1 -23039.999,E2 -23039.999} C_VEL
LIN {X 0,Y 171.818,Z 553.896,A -85,B 0,C 180,E1 -23044.692,E2 -23044.692} C_VEL
LIN {X 0,Y 171.87,Z 553.882,A -85,B 0,C 180,E1 -23049.413,E2 -23049.413} C_VEL
LIN {X 0,Y 171.59,Z 553.923,A -85,B 0,C 180,E1 -23054.225,E2 -23054.225} C_VEL
LIN {X 0,Y 171.536,Z 553.926,A -85,B 0,C 180,E1 -23059.557,E2 -23059.557} C_VEL
LIN {X 0,Y 171.455,Z 553.936,A -85,B 0,C 180,E1 -23065.609,E2 -23065.609} C_VEL
LIN {X 0,Y 171.455,Z 553.94,A -85,B 0,C 180,E1 -23070.596,E2 -23070.596} C_VEL
LIN {X 0,Y 171.39,Z 553.943,A -85,B 0,C 180,E1 -23075.035,E2 -23075.035} C_VEL
LIN {X 0,Y 171.354,Z 553.953,A -85,B 0,C 180,E1 -23078.807,E2 -23078.807} C_VEL
LIN {X 0,Y 171.323,Z 553.955,A -85,B 0,C 180,E1 -23084.216,E2 -23084.216} C_VEL
LIN {X 0,Y 171.381,Z 553.95,A -85,B 0,C 180,E1 -23088.996,E2 -23088.996} C_VEL
LIN {X 0,Y 171.956,Z 554.04,A -85,B 0,C 180,E1 -23094.423,E2 -23094.423} C_VEL
LIN {X 0,Y 173.771,Z 561.923,A -85,B 0,C 180,E1 -23099.03,E2 -23099.03} C_VEL
LIN {X 0,Y 173.811,Z 564.216,A -85,B 0,C 180,E1 -23100.333,E2 -23100.333} C_VEL
LIN {X 0,Y 173.308,Z 566.678,A -85,B 0,C 180,E1 -23101.541,E2 -23101.541} C_VEL
LIN {X 0,Y 173.32,Z 590.238,A -85,B 0,C 180,E1 -23103.207,E2 -23103.207} C_VEL
LIN {X 0,Y 175.128,Z 632.96,A -85,B 0,C 180,E1 -23106.223,E2 -23106.223} C_VEL
LIN {X 0,Y 176.37,Z 655.851,A -85,B 0,C 180,E1 -23107.914,E2 -23107.914} C_VEL
LIN {X 0,Y 175.656,Z 667.945,A -85,B 0,C 180,E1 -23109.201,E2 -23109.201} C_VEL
LIN {X 0,Y 174.727,Z 679.718,A -85,B 0,C 180,E1 -23110.925,E2 -23110.925} C_VEL
LIN {X 0,Y 173.416,Z 691.422,A -85,B 0,C 180,E1 -23113.217,E2 -23113.217} C_VEL
LIN {X 0,Y 172.413,Z 701.712,A -85,B 0,C 180,E1 -23115.843,E2 -23115.843} C_VEL
LIN {X 0,Y 171.733,Z 710.668,A -85,B 0,C 180,E1 -23118.757,E2 -23118.757} C_VEL
LIN {X 0,Y 171.523,Z 717.983,A -85,B 0,C 180,E1 -23121.755,E2 -23121.755} C_VEL
LIN {X 0,Y 171.876,Z 724.716,A -85,B 0,C 180,E1 -23125.309,E2 -23125.309} C_VEL
LIN {X 0,Y 172.592,Z 729.726,A -85,B 0,C 180,E1 -23128.833,E2 -23128.833} C_VEL
LIN {X 0,Y 172.796,Z 731.035,A -85,B 0,C 180,E1 -23130.029,E2 -23130.029} C_VEL
LIN {X 0,Y 171.39,Z 732.32,A -85,B 0,C 180,E1 -23131.896,E2 -23131.896} C_VEL
LIN {X 0,Y 167.585,Z 733.333,A -85,B 0,C 180,E1 -23134.974,E2 -23134.974} C_VEL
LIN {X 0,Y 164.703,Z 733.659,A -85,B 0,C 180,E1 -23137.545,E2 -23137.545} C_VEL
LIN {X 0,Y 163.526,Z 733.724,A -85,B 0,C 180,E1 -23139.583,E2 -23139.583} C_VEL
LIN {X 0,Y 163.444,Z 733.727,A -85,B 0,C 180,E1 -23140.278,E2 -23140.278} C_VEL
LIN {X 0,Y 164.142,Z 733.324,A -85,B 0,C 180,E1 -23144.886,E2 -23144.886} C_VEL
LIN {X 0,Y 165.13,Z 732.536,A -85,B 0,C 180,E1 -23147.332,E2 -23147.332} C_VEL
LIN {X 0,Y 166.626,Z 731.329,A -85,B 0,C 180,E1 -23149.719,E2 -23149.719} C_VEL
LIN {X 0,Y 169.557,Z 728.721,A -85,B 0,C 180,E1 -23153.188,E2 -23153.188} C_VEL
LIN {X 0,Y 174.293,Z 724.163,A -85,B 0,C 180,E1 -23157.236,E2 -23157.236} C_VEL
LIN {X 0,Y 179.54,Z 718.648,A -85,B 0,C 180,E1 -23160.588,E2 -23160.588} C_VEL
LIN {X 0,Y 186.095,Z 711.175,A -85,B 0,C 180,E1 -23163.85,E2 -23163.85} C_VEL
LIN {X 0,Y 192.332,Z 703.094,A -85,B 0,C 180,E1 -23166.425,E2 -23166.425} C_VEL
LIN {X 0,Y 197.987,Z 694.895,A -85,B 0,C 180,E1 -23168.403,E2 -23168.403} C_VEL
LIN {X 0,Y 204.063,Z 685.092,A -85,B 0,C 180,E1 -23170.221,E2 -23170.221} C_VEL
LIN {X 0,Y 209.906,Z 674.199,A -85,B 0,C 180,E1 -23171.715,E2 -23171.715} C_VEL
LIN {X 0,Y 214.334,Z 664.033,A -85,B 0,C 180,E1 -23172.873,E2 -23172.873} C_VEL
LIN {X 0,Y 218.671,Z 650.806,A -85,B 0,C 180,E1 -23174.283,E2 -23174.283} C_VEL
LIN {X 0,Y 221.204,Z 639.012,A -85,B 0,C 180,E1 -23175.656,E2 -23175.656} C_VEL
LIN {X 0,Y 222.59,Z 627.531,A -85,B 0,C 180,E1 -23177.159,E2 -23177.159} C_VEL
LIN {X 0,Y 222.615,Z 625.853,A -85,B 0,C 180,E1 -23177.534,E2 -23177.534} C_VEL
LIN {X 0,Y 222.179,Z 620.543,A -85,B 0,C 180,E1 -23179.389,E2 -23179.389} C_VEL
LIN {X 0,Y 222.041,Z 619.287,A -85,B 0,C 180,E1 -23179.911,E2 -23179.911} C_VEL
LIN {X 0,Y 220.968,Z 615.937,A -85,B 0,C 180,E1 -23184.398,E2 -23184.398} C_VEL
LIN {X 0,Y 221.008,Z 616.053,A -85,B 0,C 180,E1 -23187.276,E2 -23187.276} C_VEL
LIN {X 0,Y 222.244,Z 619.841,A -85,B 0,C 180,E1 -23192.1,E2 -23192.1} C_VEL
LIN {X 0,Y 223.353,Z 623.341,A -85,B 0,C 180,E1 -23194.701,E2 -23194.701} C_VEL
LIN {X 0,Y 224.304,Z 627.151,A -85,B 0,C 180,E1 -23196.864,E2 -23196.864} C_VEL
LIN {X 0,Y 224.032,Z 628.906,A -85,B 0,C 180,E1 -23197.194,E2 -23197.194} C_VEL
LIN {X 0,Y 220.77,Z 639.137,A -85,B 0,C 180,E1 -23198.383,E2 -23198.383} C_VEL
LIN {X 0,Y 216.833,Z 648.778,A -85,B 0,C 180,E1 -23199.77,E2 -23199.77} C_VEL
LIN {X 0,Y 211.819,Z 658.825,A -85,B 0,C 180,E1 -23201.628,E2 -23201.628} C_VEL
LIN {X 0,Y 206.178,Z 668.137,A -85,B 0,C 180,E1 -23203.854,E2 -23203.854} C_VEL
LIN {X 0,Y 200.496,Z 675.858,A -85,B 0,C 180,E1 -23206.314,E2 -23206.314} C_VEL
LIN {X 0,Y 195.569,Z 681.445,A -85,B 0,C 180,E1 -23208.601,E2 -23208.601} C_VEL
LIN {X 0,Y 190.134,Z 686.764,A -85,B 0,C 180,E1 -23211.498,E2 -23211.498} C_VEL
LIN {X 0,Y 185.062,Z 690.734,A -85,B 0,C 180,E1 -23214.553,E2 -23214.553} C_VEL
LIN {X 0,Y 180.517,Z 693.459,A -85,B 0,C 180,E1 -23217.77,E2 -23217.77} C_VEL
LIN {X 0,Y 175.783,Z 695.309,A -85,B 0,C 180,E1 -23221.807,E2 -23221.807} C_VEL
LIN {X 0,Y 172.983,Z 695.672,A -85,B 0,C 180,E1 -23224.662,E2 -23224.662} C_VEL
LIN {X 0,Y 170.299,Z 695.27,A -85,B 0,C 180,E1 -23227.938,E2 -23227.938} C_VEL
LIN {X 0,Y 167.696,Z 693.6,A -85,B 0,C 180,E1 -23232.097,E2 -23232.097} C_VEL
LIN {X 0,Y 166.037,Z 690.883,A -85,B 0,C 180,E1 -23235.971,E2 -23235.971} C_VEL
LIN {X 0,Y 164.885,Z 686.478,A -85,B 0,C 180,E1 -23240.332,E2 -23240.332} C_VEL
LIN {X 0,Y 164.536,Z 680.673,A -85,B 0,C 180,E1 -23244.612,E2 -23244.612} C_VEL
LIN {X 0,Y 164.876,Z 673.567,A -85,B 0,C 180,E1 -23248.657,E2 -23248.657} C_VEL
LIN {X 0,Y 165.457,Z 666.615,A -85,B 0,C 180,E1 -23251.843,E2 -23251.843} C_VEL
LIN {X 0,Y 166.487,Z 657.828,A -85,B 0,C 180,E1 -23255.112,E2 -23255.112} C_VEL
LIN {X 0,Y 167.743,Z 647.013,A -85,B 0,C 180,E1 -23258.345,E2 -23258.345} C_VEL
LIN {X 0,Y 169.028,Z 636.135,A -85,B 0,C 180,E1 -23260.911,E2 -23260.911} C_VEL
LIN {X 0,Y 170.314,Z 623.855,A -85,B 0,C 180,E1 -23263.196,E2 -23263.196} C_VEL
LIN {X 0,Y 171.441,Z 610.414,A -85,B 0,C 180,E1 -23265.073,E2 -23265.073} C_VEL
LIN {X 0,Y 172.227,Z 597.792,A -85,B 0,C 180,E1 -23266.324,E2 -23266.324} C_VEL
LIN {X 0,Y 172.663,Z 582.593,A -85,B 0,C 180,E1 -23267.355,E2 -23267.355} C_VEL
LIN {X 0,Y 164.619,Z 555.666,A -85,B 0,C 180,E1 -23269.681,E2 -23269.681} C_VEL
LIN {X 0,Y 164.44,Z 554.894,A -85,B 0,C 180,E1 -23270.129,E2 -23270.129} C_VEL
LIN {X 0,Y 164.337,Z 554.827,A -85,B 0,C 180,E1 -23276.225,E2 -23276.225} C_VEL
LIN {X 0,Y 164.408,Z 554.819,A -85,B 0,C 180,E1 -23279.139,E2 -23279.139} C_VEL
LIN {X 0,Y 164.419,Z 554.816,A -85,B 0,C 180,E1 -23284.695,E2 -23284.695} C_VEL
LIN {X 0,Y 164.487,Z 554.807,A -85,B 0,C 180,E1 -23290.052,E2 -23290.052} C_VEL
LIN {X 0,Y 164.502,Z 554.802,A -85,B 0,C 180,E1 -23295.148,E2 -23295.148} C_VEL
LIN {X 0,Y 164.77,Z 554.77,A -85,B 0,C 180,E1 -23300.177,E2 -23300.177} C_VEL
LIN {X 0,Y 164.83,Z 554.758,A -85,B 0,C 180,E1 -23302.651,E2 -23302.651} C_VEL
LIN {X 0,Y 165.049,Z 554.739,A -85,B 0,C 180,E1 -23307.56,E2 -23307.56} C_VEL
LIN {X 0,Y 165.299,Z 554.703,A -85,B 0,C 180,E1 -23310,E2 -23310} C_VEL
LIN {X 0,Y 164.763,Z 554.772,A -85,B 0,C 180,E1 -23314.894,E2 -23314.894} C_VEL
LIN {X 0,Y 164.831,Z 554.765,A -85,B 0,C 180,E1 -23317.349,E2 -23317.349} C_VEL
LIN {X 0,Y 164.706,Z 554.775,A -85,B 0,C 180,E1 -23321.06,E2 -23321.06} C_VEL
LIN {X 0,Y 164.487,Z 554.806,A -85,B 0,C 180,E1 -23327.403,E2 -23327.403} C_VEL
LIN {X 0,Y 164.476,Z 554.805,A -85,B 0,C 180,E1 -23329.988,E2 -23329.988} C_VEL
LIN {X 0,Y 164.388,Z 554.818,A -85,B 0,C 180,E1 -23336.127,E2 -23336.127} C_VEL
LIN {X 0,Y 164.377,Z 554.82,A -85,B 0,C 180,E1 -23341.226,E2 -23341.226} C_VEL
LIN {X 0,Y 164.349,Z 554.818,A -85,B 0,C 180,E1 -23346.774,E2 -23346.774} C_VEL
LIN {X 0,Y 164.37,Z 554.822,A -85,B 0,C 180,E1 -23349.892,E2 -23349.892} C_VEL
LIN {X 0,Y 164.341,Z 554.824,A -85,B 0,C 180,E1 -23353.363,E2 -23353.363} C_VEL
LIN {X 0,Y 164.322,Z 554.825,A -85,B 0,C 180,E1 -23356.817,E2 -23356.817} C_VEL
LIN {X 0,Y 164.308,Z 554.831,A -85,B 0,C 180,E1 -23360.345,E2 -23360.345} C_VEL
LIN {X 0,Y 164.343,Z 554.821,A -85,B 0,C 180,E1 -23364.341,E2 -23364.341} C_VEL
LIN {X 0,Y 164.39,Z 554.819,A -85,B 0,C 180,E1 -23369.133,E2 -23369.133} C_VEL
LIN {X 0,Y 164.417,Z 554.814,A -85,B 0,C 180,E1 -23374.693,E2 -23374.693} C_VEL
LIN {X 0,Y 164.501,Z 554.806,A -85,B 0,C 180,E1 -23380.033,E2 -23380.033} C_VEL
LIN {X 0,Y 164.529,Z 554.801,A -85,B 0,C 180,E1 -23385.149,E2 -23385.149} C_VEL
LIN {X 0,Y 164.82,Z 554.764,A -85,B 0,C 180,E1 -23390.179,E2 -23390.179} C_VEL
LIN {X 0,Y 164.851,Z 554.76,A -85,B 0,C 180,E1 -23392.651,E2 -23392.651} C_VEL
LIN {X 0,Y 165.047,Z 554.736,A -85,B 0,C 180,E1 -23397.559,E2 -23397.559} C_VEL
LIN {X 0,Y 165.292,Z 554.703,A -85,B 0,C 180,E1 -23399.999,E2 -23399.999} C_VEL
LIN {X 0,Y 164.767,Z 554.773,A -85,B 0,C 180,E1 -23404.893,E2 -23404.893} C_VEL
LIN {X 0,Y 164.842,Z 554.76,A -85,B 0,C 180,E1 -23407.348,E2 -23407.348} C_VEL
LIN {X 0,Y 164.747,Z 554.774,A -85,B 0,C 180,E1 -23411.145,E2 -23411.145} C_VEL
LIN {X 0,Y 164.48,Z 554.803,A -85,B 0,C 180,E1 -23417.403,E2 -23417.403} C_VEL
LIN {X 0,Y 164.47,Z 554.807,A -85,B 0,C 180,E1 -23419.989,E2 -23419.989} C_VEL
LIN {X 0,Y 164.383,Z 554.817,A -85,B 0,C 180,E1 -23426.128,E2 -23426.128} C_VEL
LIN {X 0,Y 164.385,Z 554.82,A -85,B 0,C 180,E1 -23431.235,E2 -23431.235} C_VEL
LIN {X 0,Y 164.291,Z 554.828,A -85,B 0,C 180,E1 -23436.789,E2 -23436.789} C_VEL
LIN {X 0,Y 164.288,Z 554.832,A -85,B 0,C 180,E1 -23439.916,E2 -23439.916} C_VEL
LIN {X 0,Y 164.277,Z 554.833,A -85,B 0,C 180,E1 -23443.342,E2 -23443.342} C_VEL
LIN {X 0,Y 164.29,Z 554.833,A -85,B 0,C 180,E1 -23446.809,E2 -23446.809} C_VEL
LIN {X 0,Y 164.942,Z 554.837,A -85,B 0,C 180,E1 -23454.692,E2 -23454.692} C_VEL
LIN {X 0,Y 166.812,Z 562.816,A -85,B 0,C 180,E1 -23459.631,E2 -23459.631} C_VEL
LIN {X 0,Y 166.456,Z 565.059,A -85,B 0,C 180,E1 -23460.866,E2 -23460.866} C_VEL
LIN {X 0,Y 166.266,Z 568.719,A -85,B 0,C 180,E1 -23461.262,E2 -23461.262} C_VEL
LIN {X 0,Y 166.555,Z 599.356,A -85,B 0,C 180,E1 -23463.448,E2 -23463.448} C_VEL
LIN {X 0,Y 169.216,Z 653.998,A -85,B 0,C 180,E1 -23467.546,E2 -23467.546} C_VEL
LIN {X 0,Y 168.857,Z 662.979,A -85,B 0,C 180,E1 -23468.483,E2 -23468.483} C_VEL
LIN {X 0,Y 168.023,Z 674.833,A -85,B 0,C 180,E1 -23470.133,E2 -23470.133} C_VEL
LIN {X 0,Y 166.898,Z 686.068,A -85,B 0,C 180,E1 -23472.224,E2 -23472.224} C_VEL
LIN {X 0,Y 165.659,Z 697.179,A -85,B 0,C 180,E1 -23474.939,E2 -23474.939} C_VEL
LIN {X 0,Y 165.015,Z 706.073,A -85,B 0,C 180,E1 -23477.705,E2 -23477.705} C_VEL
LIN {X 0,Y 164.6,Z 713.969,A -85,B 0,C 180,E1 -23480.786,E2 -23480.786} C_VEL
LIN {X 0,Y 164.793,Z 721.392,A -85,B 0,C 180,E1 -23484.494,E2 -23484.494} C_VEL
LIN {X 0,Y 165.384,Z 726.182,A -85,B 0,C 180,E1 -23487.564,E2 -23487.564} C_VEL
LIN {X 0,Y 165.888,Z 729.139,A -85,B 0,C 180,E1 -23490,E2 -23490} C_VEL
LIN {X 0,Y 165.036,Z 731.085,A -85,B 0,C 180,E1 -23492.44,E2 -23492.44} C_VEL
LIN {X 0,Y 164.189,Z 732.408,A -85,B 0,C 180,E1 -23494.911,E2 -23494.911} C_VEL
LIN {X 0,Y 163.496,Z 733.545,A -85,B 0,C 180,E1 -23498.637,E2 -23498.637} C_VEL
LIN {X 0,Y 163.444,Z 733.727,A -85,B 0,C 180,E1 -23500.278,E2 -23500.278} C_VEL
LIN {X 0,Y 162.951,Z 733.633,A -85,B 0,C 180,E1 -23502.345,E2 -23502.345} C_VEL
LIN {X 0,Y 160.954,Z 732.701,A -85,B 0,C 180,E1 -23505.769,E2 -23505.769} C_VEL
LIN {X 0,Y 159.747,Z 731.222,A -85,B 0,C 180,E1 -23509.231,E2 -23509.231} C_VEL
LIN {X 0,Y 160.479,Z 730.112,A -85,B 0,C 180,E1 -23511.279,E2 -23511.279} C_VEL
LIN {X 0,Y 161.89,Z 729.092,A -85,B 0,C 180,E1 -23512.998,E2 -23512.998} C_VEL
LIN {X 0,Y 165.613,Z 726.134,A -85,B 0,C 180,E1 -23516.46,E2 -23516.46} C_VEL
LIN {X 0,Y 170.041,Z 722.145,A -85,B 0,C 180,E1 -23519.733,E2 -23519.733} C_VEL
LIN {X 0,Y 175.331,Z 717.078,A -85,B 0,C 180,E1 -23522.76,E2 -23522.76} C_VEL
LIN {X 0,Y 181.299,Z 710.736,A -85,B 0,C 180,E1 -23525.553,E2 -23525.553} C_VEL
LIN {X 0,Y 188.547,Z 702.047,A -85,B 0,C 180,E1 -23528.381,E2 -23528.381} C_VEL
LIN {X 0,Y 194.975,Z 693.373,A -85,B 0,C 180,E1 -23530.451,E2 -23530.451} C_VEL
LIN {X 0,Y 201.384,Z 683.482,A -85,B 0,C 180,E1 -23532.204,E2 -23532.204} C_VEL
LIN {X 0,Y 208.13,Z 671.305,A -85,B 0,C 180,E1 -23533.806,E2 -23533.806} C_VEL
LIN {X 0,Y 213.451,Z 658.905,A -85,B 0,C 180,E1 -23535.213,E2 -23535.213} C_VEL
LIN {X 0,Y 216.768,Z 648.564,A -85,B 0,C 180,E1 -23536.363,E2 -23536.363} C_VEL
LIN {X 0,Y 219.639,Z 635.528,A -85,B 0,C 180,E1 -23538.022,E2 -23538.022} C_VEL
LIN {X 0,Y 220.369,Z 630.672,A -85,B 0,C 180,E1 -23538.756,E2 -23538.756} C_VEL
LIN {X 0,Y 220.262,Z 625.893,A -85,B 0,C 180,E1 -23540.528,E2 -23540.528} C_VEL
LIN {X 0,Y 219.446,Z 622.81,A -85,B 0,C 180,E1 -23544.798,E2 -23544.798} C_VEL
LIN {X 0,Y 219.365,Z 622.903,A -85,B 0,C 180,E1 -23547,E2 -23547} C_VEL
LIN {X 0,Y 219.967,Z 626.001,A -85,B 0,C 180,E1 -23551.364,E2 -23551.364} C_VEL
LIN {X 0,Y 220.904,Z 630.654,A -85,B 0,C 180,E1 -23554.903,E2 -23554.903} C_VEL
LIN {X 0,Y 221.079,Z 631.82,A -85,B 0,C 180,E1 -23555.591,E2 -23555.591} C_VEL
LIN {X 0,Y 218.893,Z 638.473,A -85,B 0,C 180,E1 -23556.442,E2 -23556.442} C_VEL
LIN {X 0,Y 214.252,Z 649.661,A -85,B 0,C 180,E1 -23557.981,E2 -23557.981} C_VEL
LIN {X 0,Y 209.034,Z 659.733,A -85,B 0,C 180,E1 -23559.791,E2 -23559.791} C_VEL
LIN {X 0,Y 203.327,Z 668.623,A -85,B 0,C 180,E1 -23561.876,E2 -23561.876} C_VEL
LIN {X 0,Y 197.561,Z 676.217,A -85,B 0,C 180,E1 -23564.193,E2 -23564.193} C_VEL
LIN {X 0,Y 191.72,Z 682.608,A -85,B 0,C 180,E1 -23566.756,E2 -23566.756} C_VEL
LIN {X 0,Y 185.694,Z 688.056,A -85,B 0,C 180,E1 -23569.737,E2 -23569.737} C_VEL
LIN {X 0,Y 179.509,Z 692.462,A -85,B 0,C 180,E1 -23573.256,E2 -23573.256} C_VEL
LIN {X 0,Y 176.256,Z 694.324,A -85,B 0,C 180,E1 -23575.427,E2 -23575.427} C_VEL
LIN {X 0,Y 173.185,Z 695.657,A -85,B 0,C 180,E1 -23577.675,E2 -23577.675} C_VEL
LIN {X 0,Y 168.727,Z 696.809,A -85,B 0,C 180,E1 -23581.527,E2 -23581.527} C_VEL
LIN {X 0,Y 165.505,Z 696.815,A -85,B 0,C 180,E1 -23584.873,E2 -23584.873} C_VEL
LIN {X 0,Y 163.152,Z 696.138,A -85,B 0,C 180,E1 -23587.808,E2 -23587.808} C_VEL
LIN {X 0,Y 160.239,Z 693.701,A -85,B 0,C 180,E1 -23592.669,E2 -23592.669} C_VEL
LIN {X 0,Y 158.649,Z 690.448,A -85,B 0,C 180,E1 -23596.736,E2 -23596.736} C_VEL
LIN {X 0,Y 157.699,Z 685.918,A -85,B 0,C 180,E1 -23600.888,E2 -23600.888} C_VEL
LIN {X 0,Y 157.441,Z 679.981,A -85,B 0,C 180,E1 -23605.093,E2 -23605.093} C_VEL
LIN {X 0,Y 157.875,Z 672.342,A -85,B 0,C 180,E1 -23609.321,E2 -23609.321} C_VEL
LIN {X 0,Y 158.663,Z 664.049,A -85,B 0,C 180,E1 -23612.995,E2 -23612.995} C_VEL
LIN {X 0,Y 159.775,Z 654.365,A -85,B 0,C 180,E1 -23616.43,E2 -23616.43} C_VEL
LIN {X 0,Y 160.973,Z 644.443,A -85,B 0,C 180,E1 -23619.276,E2 -23619.276} C_VEL
LIN {X 0,Y 162.254,Z 633.695,A -85,B 0,C 180,E1 -23621.729,E2 -23621.729} C_VEL
LIN {X 0,Y 163.484,Z 621.719,A -85,B 0,C 180,E1 -23623.885,E2 -23623.885} C_VEL
LIN {X 0,Y 164.465,Z 610.001,A -85,B 0,C 180,E1 -23625.489,E2 -23625.489} C_VEL
LIN {X 0,Y 165.315,Z 596.31,A -85,B 0,C 180,E1 -23626.831,E2 -23626.831} C_VEL
LIN {X 0,Y 165.512,Z 583.285,A -85,B 0,C 180,E1 -23627.721,E2 -23627.721} C_VEL
LIN {X 0,Y 157.543,Z 556.495,A -85,B 0,C 180,E1 -23630.161,E2 -23630.161} C_VEL
LIN {X 0,Y 157.359,Z 555.774,A -85,B 0,C 180,E1 -23630.619,E2 -23630.619} C_VEL
LIN {X 0,Y 157.294,Z 555.704,A -85,B 0,C 180,E1 -23634.491,E2 -23634.491} C_VEL
LIN {X 0,Y 157.304,Z 555.703,A -85,B 0,C 180,E1 -23638.092,E2 -23638.092} C_VEL
LIN {X 0,Y 157.325,Z 555.701,A -85,B 0,C 180,E1 -23643.468,E2 -23643.468} C_VEL
LIN {X 0,Y 157.397,Z 555.692,A -85,B 0,C 180,E1 -23649.669,E2 -23649.669} C_VEL
LIN {X 0,Y 157.439,Z 555.681,A -85,B 0,C 180,E1 -23654.465,E2 -23654.465} C_VEL
LIN {X 0,Y 157.692,Z 555.654,A -85,B 0,C 180,E1 -23659.731,E2 -23659.731} C_VEL
LIN {X 0,Y 157.768,Z 555.638,A -85,B 0,C 180,E1 -23662.32,E2 -23662.32} C_VEL
LIN {X 0,Y 158.261,Z 555.579,A -85,B 0,C 180,E1 -23670,E2 -23670} C_VEL
LIN {X 0,Y 157.768,Z 555.645,A -85,B 0,C 180,E1 -23677.68,E2 -23677.68} C_VEL
LIN {X 0,Y 157.641,Z 555.655,A -85,B 0,C 180,E1 -23681.236,E2 -23681.236} C_VEL
LIN {X 0,Y 157.457,Z 555.684,A -85,B 0,C 180,E1 -23685.534,E2 -23685.534} C_VEL
LIN {X 0,Y 157.371,Z 555.691,A -85,B 0,C 180,E1 -23690.932,E2 -23690.932} C_VEL
LIN {X 0,Y 157.312,Z 555.697,A -85,B 0,C 180,E1 -23696.68,E2 -23696.68} C_VEL
LIN {X 0,Y 157.279,Z 555.706,A -85,B 0,C 180,E1 -23702.426,E2 -23702.426} C_VEL
LIN {X 0,Y 157.324,Z 555.694,A -85,B 0,C 180,E1 -23706.475,E2 -23706.475} C_VEL
LIN {X 0,Y 157.272,Z 555.708,A -85,B 0,C 180,E1 -23712.09,E2 -23712.09} C_VEL
LIN {X 0,Y 157.232,Z 555.709,A -85,B 0,C 180,E1 -23717.895,E2 -23717.895} C_VEL
LIN {X 0,Y 157.283,Z 555.702,A -85,B 0,C 180,E1 -23723.542,E2 -23723.542} C_VEL
LIN {X 0,Y 157.294,Z 555.704,A -85,B 0,C 180,E1 -23728.094,E2 -23728.094} C_VEL
LIN {X 0,Y 157.321,Z 555.694,A -85,B 0,C 180,E1 -23733.465,E2 -23733.465} C_VEL
LIN {X 0,Y 157.417,Z 555.688,A -85,B 0,C 180,E1 -23739.643,E2 -23739.643} C_VEL
LIN {X 0,Y 157.461,Z 555.681,A -85,B 0,C 180,E1 -23744.466,E2 -23744.466} C_VEL
LIN {X 0,Y 157.736,Z 555.646,A -85,B 0,C 180,E1 -23749.733,E2 -23749.733} C_VEL
LIN {X 0,Y 157.811,Z 555.634,A -85,B 0,C 180,E1 -23752.321,E2 -23752.321} C_VEL
LIN {X 0,Y 158.254,Z 555.58,A -85,B 0,C 180,E1 -23759.999,E2 -23759.999} C_VEL
LIN {X 0,Y 157.8,Z 555.638,A -85,B 0,C 180,E1 -23767.677,E2 -23767.677} C_VEL
LIN {X 0,Y 157.677,Z 555.654,A -85,B 0,C 180,E1 -23771.314,E2 -23771.314} C_VEL
LIN {X 0,Y 157.457,Z 555.682,A -85,B 0,C 180,E1 -23775.533,E2 -23775.533} C_VEL
LIN {X 0,Y 157.364,Z 555.696,A -85,B 0,C 180,E1 -23780.933,E2 -23780.933} C_VEL
LIN {X 0,Y 157.306,Z 555.698,A -85,B 0,C 180,E1 -23786.68,E2 -23786.68} C_VEL
LIN {X 0,Y 157.278,Z 555.706,A -85,B 0,C 180,E1 -23792.426,E2 -23792.426} C_VEL
LIN {X 0,Y 157.265,Z 555.702,A -85,B 0,C 180,E1 -23796.449,E2 -23796.449} C_VEL
LIN {X 0,Y 157.208,Z 555.713,A -85,B 0,C 180,E1 -23802.111,E2 -23802.111} C_VEL
LIN {X 0,Y 157.23,Z 555.711,A -85,B 0,C 180,E1 -23807.897,E2 -23807.897} C_VEL
LIN {X 0,Y 158.014,Z 555.719,A -85,B 0,C 180,E1 -23815.166,E2 -23815.166} C_VEL
LIN {X 0,Y 159.633,Z 562.537,A -85,B 0,C 180,E1 -23819.583,E2 -23819.583} C_VEL
LIN {X 0,Y 159.518,Z 564.27,A -85,B 0,C 180,E1 -23820.379,E2 -23820.379} C_VEL
LIN {X 0,Y 159.297,Z 588.697,A -85,B 0,C 180,E1 -23822.251,E2 -23822.251} C_VEL
LIN {X 0,Y 160.964,Z 632.87,A -85,B 0,C 180,E1 -23825.666,E2 -23825.666} C_VEL
LIN {X 0,Y 162.142,Z 654.679,A -85,B 0,C 180,E1 -23827.46,E2 -23827.46} C_VEL
LIN {X 0,Y 161.561,Z 665.922,A -85,B 0,C 180,E1 -23828.802,E2 -23828.802} C_VEL
LIN {X 0,Y 160.776,Z 676.785,A -85,B 0,C 180,E1 -23830.53,E2 -23830.53} C_VEL
LIN {X 0,Y 159.625,Z 687.26,A -85,B 0,C 180,E1 -23832.711,E2 -23832.711} C_VEL
LIN {X 0,Y 158.507,Z 697.897,A -85,B 0,C 180,E1 -23835.558,E2 -23835.558} C_VEL
LIN {X 0,Y 157.89,Z 707.055,A -85,B 0,C 180,E1 -23838.68,E2 -23838.68} C_VEL
LIN {X 0,Y 157.7,Z 715.368,A -85,B 0,C 180,E1 -23842.317,E2 -23842.317} C_VEL
LIN {X 0,Y 158.033,Z 721.202,A -85,B 0,C 180,E1 -23845.536,E2 -23845.536} C_VEL
LIN {X 0,Y 158.702,Z 725.739,A -85,B 0,C 180,E1 -23848.731,E2 -23848.731} C_VEL
LIN {X 0,Y 158.971,Z 727.21,A -85,B 0,C 180,E1 -23850,E2 -23850} C_VEL
LIN {X 0,Y 158.145,Z 729.256,A -85,B 0,C 180,E1 -23852.547,E2 -23852.547} C_VEL
LIN {X 0,Y 157.26,Z 730.727,A -85,B 0,C 180,E1 -23855.128,E2 -23855.128} C_VEL
LIN {X 0,Y 156.546,Z 732.073,A -85,B 0,C 180,E1 -23859.012,E2 -23859.012} C_VEL
LIN {X 0,Y 156.69,Z 732.456,A -85,B 0,C 180,E1 -23862.959,E2 -23862.959} C_VEL
LIN {X 0,Y 157.297,Z 732.22,A -85,B 0,C 180,E1 -23865.549,E2 -23865.549} C_VEL
LIN {X 0,Y 158.373,Z 731.56,A -85,B 0,C 180,E1 -23868.097,E2 -23868.097} C_VEL
LIN {X 0,Y 160.479,Z 730.112,A -85,B 0,C 180,E1 -23871.279,E2 -23871.279} C_VEL
LIN {X 0,Y 161.491,Z 728.881,A -85,B 0,C 180,E1 -23873.305,E2 -23873.305} C_VEL
LIN {X 0,Y 162.217,Z 725.101,A -85,B 0,C 180,E1 -23878.037,E2 -23878.037} C_VEL
LIN {X 0,Y 163.703,Z 722.487,A -85,B 0,C 180,E1 -23880.593,E2 -23880.593} C_VEL
LIN {X 0,Y 165.234,Z 721.021,A -85,B 0,C 180,E1 -23881.744,E2 -23881.744} C_VEL
LIN {X 0,Y 171.407,Z 715.53,A -85,B 0,C 180,E1 -23885.03,E2 -23885.03} C_VEL
LIN {X 0,Y 178.315,Z 708.72,A -85,B 0,C 180,E1 -23887.977,E2 -23887.977} C_VEL
LIN {X 0,Y 184.71,Z 701.506,A -85,B 0,C 180,E1 -23890.302,E2 -23890.302} C_VEL
LIN {X 0,Y 192.254,Z 691.904,A -85,B 0,C 180,E1 -23892.552,E2 -23892.552} C_VEL
LIN {X 0,Y 198.991,Z 682.131,A -85,B 0,C 180,E1 -23894.228,E2 -23894.228} C_VEL
LIN {X 0,Y 205.963,Z 670.043,A -85,B 0,C 180,E1 -23895.771,E2 -23895.771} C_VEL
LIN {X 0,Y 212.207,Z 655.769,A -85,B 0,C 180,E1 -23897.411,E2 -23897.411} C_VEL
LIN {X 0,Y 215.449,Z 645.841,A -85,B 0,C 180,E1 -23898.612,E2 -23898.612} C_VEL
LIN {X 0,Y 217.993,Z 635.105,A -85,B 0,C 180,E1 -23900.087,E2 -23900.087} C_VEL
LIN {X 0,Y 218.125,Z 632.337,A -85,B 0,C 180,E1 -23901.241,E2 -23901.241} C_VEL
LIN {X 0,Y 217.583,Z 629.653,A -85,B 0,C 180,E1 -23904.879,E2 -23904.879} C_VEL
LIN {X 0,Y 217.411,Z 629.658,A -85,B 0,C 180,E1 -23906.665,E2 -23906.665} C_VEL
LIN {X 0,Y 217.507,Z 632.539,A -85,B 0,C 180,E1 -23911.01,E2 -23911.01} C_VEL
LIN {X 0,Y 217.852,Z 636.403,A -85,B 0,C 180,E1 -23914.133,E2 -23914.133} C_VEL
LIN {X 0,Y 217.39,Z 638.024,A -85,B 0,C 180,E1 -23914.468,E2 -23914.468} C_VEL
LIN {X 0,Y 212.904,Z 648.741,A -85,B 0,C 180,E1 -23915.856,E2 -23915.856} C_VEL
LIN {X 0,Y 207.625,Z 658.752,A -85,B 0,C 180,E1 -23917.548,E2 -23917.548} C_VEL
LIN {X 0,Y 201.596,Z 668.197,A -85,B 0,C 180,E1 -23919.598,E2 -23919.598} C_VEL
LIN {X 0,Y 195.789,Z 675.657,A -85,B 0,C 180,E1 -23921.695,E2 -23921.695} C_VEL
LIN {X 0,Y 190.117,Z 681.817,A -85,B 0,C 180,E1 -23923.968,E2 -23923.968} C_VEL
LIN {X 0,Y 183.79,Z 687.578,A -85,B 0,C 180,E1 -23926.737,E2 -23926.737} C_VEL
LIN {X 0,Y 178.856,Z 691.306,A -85,B 0,C 180,E1 -23929.212,E2 -23929.212} C_VEL
LIN {X 0,Y 175.937,Z 693.187,A -85,B 0,C 180,E1 -23930.806,E2 -23930.806} C_VEL
LIN {X 0,Y 171.117,Z 695.659,A -85,B 0,C 180,E1 -23933.75,E2 -23933.75} C_VEL
LIN {X 0,Y 165.81,Z 697.601,A -85,B 0,C 180,E1 -23937.572,E2 -23937.572} C_VEL
LIN {X 0,Y 161.674,Z 698.188,A -85,B 0,C 180,E1 -23941.184,E2 -23941.184} C_VEL
LIN {X 0,Y 157.99,Z 697.719,A -85,B 0,C 180,E1 -23945.105,E2 -23945.105} C_VEL
LIN {X 0,Y 155.934,Z 696.831,A -85,B 0,C 180,E1 -23947.772,E2 -23947.772} C_VEL
LIN {X 0,Y 154.189,Z 695.414,A -85,B 0,C 180,E1 -23950.506,E2 -23950.506} C_VEL
LIN {X 0,Y 152.343,Z 692.672,A -85,B 0,C 180,E1 -23954.359,E2 -23954.359} C_VEL
LIN {X 0,Y 150.948,Z 688.145,A -85,B 0,C 180,E1 -23959.022,E2 -23959.022} C_VEL
LIN {X 0,Y 150.389,Z 682.514,A -85,B 0,C 180,E1 -23963.406,E2 -23963.406} C_VEL
LIN {X 0,Y 150.588,Z 675.313,A -85,B 0,C 180,E1 -23967.822,E2 -23967.822} C_VEL
LIN {X 0,Y 151.189,Z 667.723,A -85,B 0,C 180,E1 -23971.532,E2 -23971.532} C_VEL
LIN {X 0,Y 152.234,Z 658.329,A -85,B 0,C 180,E1 -23975.246,E2 -23975.246} C_VEL
LIN {X 0,Y 153.454,Z 648.223,A -85,B 0,C 180,E1 -23978.457,E2 -23978.457} C_VEL
LIN {X 0,Y 154.749,Z 637.492,A -85,B 0,C 180,E1 -23981.189,E2 -23981.189} C_VEL
LIN {X 0,Y 156.17,Z 625.069,A -85,B 0,C 180,E1 -23983.665,E2 -23983.665} C_VEL
LIN {X 0,Y 157.291,Z 611.97,A -85,B 0,C 180,E1 -23985.637,E2 -23985.637} C_VEL
LIN {X 0,Y 158.241,Z 597.834,A -85,B 0,C 180,E1 -23987.117,E2 -23987.117} C_VEL
LIN {X 0,Y 158.549,Z 584.631,A -85,B 0,C 180,E1 -23988.06,E2 -23988.06} C_VEL
LIN {X 0,Y 150.511,Z 557.613,A -85,B 0,C 180,E1 -23990.6,E2 -23990.6} C_VEL
LIN {X 0,Y 150.311,Z 556.685,A -85,B 0,C 180,E1 -23991.077,E2 -23991.077} C_VEL
LIN {X 0,Y 150.225,Z 556.585,A -85,B 0,C 180,E1 -23997.364,E2 -23997.364} C_VEL
LIN {X 0,Y 150.248,Z 556.58,A -85,B 0,C 180,E1 -24002.718,E2 -24002.718} C_VEL
LIN {X 0,Y 150.354,Z 556.569,A -85,B 0,C 180,E1 -24009.209,E2 -24009.209} C_VEL
LIN {X 0,Y 150.351,Z 556.564,A -85,B 0,C 180,E1 -24013.713,E2 -24013.713} C_VEL
LIN {X 0,Y 150.614,Z 556.536,A -85,B 0,C 180,E1 -24019.243,E2 -24019.243} C_VEL
LIN {X 0,Y 150.706,Z 556.519,A -85,B 0,C 180,E1 -24021.958,E2 -24021.958} C_VEL
LIN {X 0,Y 151.222,Z 556.456,A -85,B 0,C 180,E1 -24030,E2 -24030} C_VEL
LIN {X 0,Y 150.706,Z 556.522,A -85,B 0,C 180,E1 -24038.042,E2 -24038.042} C_VEL
LIN {X 0,Y 150.581,Z 556.535,A -85,B 0,C 180,E1 -24041.437,E2 -24041.437} C_VEL
LIN {X 0,Y 150.365,Z 556.566,A -85,B 0,C 180,E1 -24046.286,E2 -24046.286} C_VEL
LIN {X 0,Y 150.353,Z 556.565,A -85,B 0,C 180,E1 -24050.79,E2 -24050.79} C_VEL
LIN {X 0,Y 150.244,Z 556.578,A -85,B 0,C 180,E1 -24057.279,E2 -24057.279} C_VEL
LIN {X 0,Y 150.219,Z 556.585,A -85,B 0,C 180,E1 -24062.632,E2 -24062.632} C_VEL
LIN {X 0,Y 150.234,Z 556.576,A -85,B 0,C 180,E1 -24067.455,E2 -24067.455} C_VEL
LIN {X 0,Y 150.217,Z 556.585,A -85,B 0,C 180,E1 -24071.532,E2 -24071.532} C_VEL
LIN {X 0,Y 150.168,Z 556.586,A -85,B 0,C 180,E1 -24075.41,E2 -24075.41} C_VEL
LIN {X 0,Y 150.168,Z 556.59,A -85,B 0,C 180,E1 -24079.063,E2 -24079.063} C_VEL
LIN {X 0,Y 150.216,Z 556.583,A -85,B 0,C 180,E1 -24082.688,E2 -24082.688} C_VEL
LIN {X 0,Y 150.218,Z 556.583,A -85,B 0,C 180,E1 -24087.365,E2 -24087.365} C_VEL
LIN {X 0,Y 150.244,Z 556.576,A -85,B 0,C 180,E1 -24092.717,E2 -24092.717} C_VEL
LIN {X 0,Y 150.366,Z 556.566,A -85,B 0,C 180,E1 -24099.191,E2 -24099.191} C_VEL
LIN {X 0,Y 150.371,Z 556.561,A -85,B 0,C 180,E1 -24103.713,E2 -24103.713} C_VEL
LIN {X 0,Y 150.652,Z 556.529,A -85,B 0,C 180,E1 -24109.244,E2 -24109.244} C_VEL
LIN {X 0,Y 150.746,Z 556.513,A -85,B 0,C 180,E1 -24111.959,E2 -24111.959} C_VEL
LIN {X 0,Y 151.215,Z 556.456,A -85,B 0,C 180,E1 -24119.999,E2 -24119.999} C_VEL
LIN {X 0,Y 150.736,Z 556.518,A -85,B 0,C 180,E1 -24128.04,E2 -24128.04} C_VEL
LIN {X 0,Y 150.608,Z 556.534,A -85,B 0,C 180,E1 -24131.499,E2 -24131.499} C_VEL
LIN {X 0,Y 150.363,Z 556.566,A -85,B 0,C 180,E1 -24136.286,E2 -24136.286} C_VEL
LIN {X 0,Y 150.346,Z 556.569,A -85,B 0,C 180,E1 -24140.79,E2 -24140.79} C_VEL
LIN {X 0,Y 150.239,Z 556.577,A -85,B 0,C 180,E1 -24147.28,E2 -24147.28} C_VEL
LIN {X 0,Y 150.217,Z 556.586,A -85,B 0,C 180,E1 -24152.635,E2 -24152.635} C_VEL
LIN {X 0,Y 150.17,Z 556.589,A -85,B 0,C 180,E1 -24157.473,E2 -24157.473} C_VEL
LIN {X 0,Y 150.147,Z 556.593,A -85,B 0,C 180,E1 -24161.504,E2 -24161.504} C_VEL
LIN {X 0,Y 150.123,Z 556.597,A -85,B 0,C 180,E1 -24165.395,E2 -24165.395} C_VEL
LIN {X 0,Y 150.505,Z 556.551,A -85,B 0,C 180,E1 -24172.624,E2 -24172.624} C_VEL
LIN {X 0,Y 151.045,Z 556.557,A -85,B 0,C 180,E1 -24175.656,E2 -24175.656} C_VEL
LIN {X 0,Y 152.499,Z 562.482,A -85,B 0,C 180,E1 -24179.608,E2 -24179.608} C_VEL
LIN {X 0,Y 152.487,Z 565.786,A -85,B 0,C 180,E1 -24180.013,E2 -24180.013} C_VEL
LIN {X 0,Y 152.352,Z 590.958,A -85,B 0,C 180,E1 -24181.986,E2 -24181.986} C_VEL
LIN {X 0,Y 153.978,Z 633.979,A -85,B 0,C 180,E1 -24185.485,E2 -24185.485} C_VEL
LIN {X 0,Y 155.052,Z 654.173,A -85,B 0,C 180,E1 -24187.251,E2 -24187.251} C_VEL
LIN {X 0,Y 154.446,Z 666.379,A -85,B 0,C 180,E1 -24188.827,E2 -24188.827} C_VEL
LIN {X 0,Y 153.485,Z 678.452,A -85,B 0,C 180,E1 -24190.959,E2 -24190.959} C_VEL
LIN {X 0,Y 152.365,Z 688.391,A -85,B 0,C 180,E1 -24193.245,E2 -24193.245} C_VEL
LIN {X 0,Y 151.386,Z 698.552,A -85,B 0,C 180,E1 -24196.236,E2 -24196.236} C_VEL
LIN {X 0,Y 150.88,Z 706.688,A -85,B 0,C 180,E1 -24199.262,E2 -24199.262} C_VEL
LIN {X 0,Y 150.807,Z 713.973,A -85,B 0,C 180,E1 -24202.637,E2 -24202.637} C_VEL
LIN {X 0,Y 151.196,Z 719.814,A -85,B 0,C 180,E1 -24206.002,E2 -24206.002} C_VEL
LIN {X 0,Y 152.049,Z 725.132,A -85,B 0,C 180,E1 -24210,E2 -24210} C_VEL
LIN {X 0,Y 151.253,Z 727.385,A -85,B 0,C 180,E1 -24212.663,E2 -24212.663} C_VEL
LIN {X 0,Y 150.331,Z 728.996,A -85,B 0,C 180,E1 -24215.365,E2 -24215.365} C_VEL
LIN {X 0,Y 149.583,Z 730.829,A -85,B 0,C 180,E1 -24220.832,E2 -24220.832} C_VEL
LIN {X 0,Y 149.808,Z 731.122,A -85,B 0,C 180,E1 -24223.566,E2 -24223.566} C_VEL
LIN {X 0,Y 151.652,Z 730.54,A -85,B 0,C 180,E1 -24228.929,E2 -24228.929} C_VEL
LIN {X 0,Y 153.657,Z 729.467,A -85,B 0,C 180,E1 -24231.934,E2 -24231.934} C_VEL
LIN {X 0,Y 155.384,Z 728.393,A -85,B 0,C 180,E1 -24234.02,E2 -24234.02} C_VEL
LIN {X 0,Y 159.292,Z 725.717,A -85,B 0,C 180,E1 -24237.597,E2 -24237.597} C_VEL
LIN {X 0,Y 163.917,Z 722.082,A -85,B 0,C 180,E1 -24240.963,E2 -24240.963} C_VEL
LIN {X 0,Y 165.234,Z 721.021,A -85,B 0,C 180,E1 -24241.744,E2 -24241.744} C_VEL
LIN {X 0,Y 167.523,Z 718.711,A -85,B 0,C 180,E1 -24243.443,E2 -24243.443} C_VEL
LIN {X 0,Y 170.042,Z 714.562,A -85,B 0,C 180,E1 -24246.38,E2 -24246.38} C_VEL
LIN {X 0,Y 172.922,Z 709.893,A -85,B 0,C 180,E1 -24249.124,E2 -24249.124} C_VEL
LIN {X 0,Y 175.684,Z 706.734,A -85,B 0,C 180,E1 -24250.483,E2 -24250.483} C_VEL
LIN {X 0,Y 181.918,Z 700.152,A -85,B 0,C 180,E1 -24252.536,E2 -24252.536} C_VEL
LIN {X 0,Y 189.828,Z 690.634,A -85,B 0,C 180,E1 -24254.702,E2 -24254.702} C_VEL
LIN {X 0,Y 196.859,Z 680.865,A -85,B 0,C 180,E1 -24256.296,E2 -24256.296} C_VEL
LIN {X 0,Y 203.995,Z 669.081,A -85,B 0,C 180,E1 -24257.791,E2 -24257.791} C_VEL
LIN {X 0,Y 209.451,Z 657.608,A -85,B 0,C 180,E1 -24259.114,E2 -24259.114} C_VEL
LIN {X 0,Y 213.239,Z 647.321,A -85,B 0,C 180,E1 -24260.396,E2 -24260.396} C_VEL
LIN {X 0,Y 215.595,Z 639.655,A -85,B 0,C 180,E1 -24261.475,E2 -24261.475} C_VEL
LIN {X 0,Y 215.705,Z 638.92,A -85,B 0,C 180,E1 -24261.754,E2 -24261.754} C_VEL
LIN {X 0,Y 215.351,Z 636.628,A -85,B 0,C 180,E1 -24264.672,E2 -24264.672} C_VEL
LIN {X 0,Y 215.156,Z 636.372,A -85,B 0,C 180,E1 -24266.269,E2 -24266.269} C_VEL
LIN {X 0,Y 214.772,Z 638.919,A -85,B 0,C 180,E1 -24270.605,E2 -24270.605} C_VEL
LIN {X 0,Y 214.685,Z 641.296,A -85,B 0,C 180,E1 -24272.723,E2 -24272.723} C_VEL
LIN {X 0,Y 213.995,Z 643.228,A -85,B 0,C 180,E1 -24273.144,E2 -24273.144} C_VEL
LIN {X 0,Y 208.927,Z 653.779,A -85,B 0,C 180,E1 -24274.604,E2 -24274.604} C_VEL
LIN {X 0,Y 203.935,Z 662.36,A -85,B 0,C 180,E1 -24276.114,E2 -24276.114} C_VEL
LIN {X 0,Y 198.447,Z 670.188,A -85,B 0,C 180,E1 -24277.859,E2 -24277.859} C_VEL
LIN {X 0,Y 191.643,Z 678.248,A -85,B 0,C 180,E1 -24280.171,E2 -24280.171} C_VEL
LIN {X 0,Y 184.776,Z 685.037,A -85,B 0,C 180,E1 -24282.808,E2 -24282.808} C_VEL
LIN {X 0,Y 179.014,Z 689.696,A -85,B 0,C 180,E1 -24285.216,E2 -24285.216} C_VEL
LIN {X 0,Y 172.056,Z 694.263,A -85,B 0,C 180,E1 -24288.61,E2 -24288.61} C_VEL
LIN {X 0,Y 168.79,Z 695.999,A -85,B 0,C 180,E1 -24290.414,E2 -24290.414} C_VEL
LIN {X 0,Y 162.401,Z 698.468,A -85,B 0,C 180,E1 -24294.452,E2 -24294.452} C_VEL
LIN {X 0,Y 158.38,Z 699.303,A -85,B 0,C 180,E1 -24297.458,E2 -24297.458} C_VEL
LIN {X 0,Y 154.627,Z 699.418,A -85,B 0,C 180,E1 -24300.794,E2 -24300.794} C_VEL
LIN {X 0,Y 150.423,Z 698.36,A -85,B 0,C 180,E1 -24305.363,E2 -24305.363} C_VEL
LIN {X 0,Y 148.392,Z 697.106,A -85,B 0,C 180,E1 -24308.169,E2 -24308.169} C_VEL
LIN {X 0,Y 145.974,Z 694.271,A -85,B 0,C 180,E1 -24312.514,E2 -24312.514} C_VEL
LIN {X 0,Y 144.332,Z 690.252,A -85,B 0,C 180,E1 -24316.988,E2 -24316.988} C_VEL
LIN {X 0,Y 143.447,Z 685.082,A -85,B 0,C 180,E1 -24321.431,E2 -24321.431} C_VEL
LIN {X 0,Y 143.323,Z 678.028,A -85,B 0,C 180,E1 -24326.19,E2 -24326.19} C_VEL
LIN {X 0,Y 143.832,Z 670.908,A -85,B 0,C 180,E1 -24330.057,E2 -24330.057} C_VEL
LIN {X 0,Y 144.605,Z 662.748,A -85,B 0,C 180,E1 -24333.701,E2 -24333.701} C_VEL
LIN {X 0,Y 145.718,Z 653.373,A -85,B 0,C 180,E1 -24337.078,E2 -24337.078} C_VEL
LIN {X 0,Y 147.108,Z 642.264,A -85,B 0,C 180,E1 -24340.295,E2 -24340.295} C_VEL
LIN {X 0,Y 148.472,Z 630.901,A -85,B 0,C 180,E1 -24342.88,E2 -24342.88} C_VEL
LIN {X 0,Y 149.691,Z 618.506,A -85,B 0,C 180,E1 -24345.074,E2 -24345.074} C_VEL
LIN {X 0,Y 150.822,Z 604.382,A -85,B 0,C 180,E1 -24346.871,E2 -24346.871} C_VEL
LIN {X 0,Y 151.475,Z 590.434,A -85,B 0,C 180,E1 -24348.051,E2 -24348.051} C_VEL
LIN {X 0,Y 151.476,Z 585.69,A -85,B 0,C 180,E1 -24348.402,E2 -24348.402} C_VEL
LIN {X 0,Y 143.407,Z 558.285,A -85,B 0,C 180,E1 -24351.131,E2 -24351.131} C_VEL
LIN {X 0,Y 143.225,Z 557.504,A -85,B 0,C 180,E1 -24351.733,E2 -24351.733} C_VEL
LIN {X 0,Y 143.192,Z 557.461,A -85,B 0,C 180,E1 -24357.325,E2 -24357.325} C_VEL
LIN {X 0,Y 143.195,Z 557.459,A -85,B 0,C 180,E1 -24362.063,E2 -24362.063} C_VEL
LIN {X 0,Y 143.279,Z 557.449,A -85,B 0,C 180,E1 -24368.747,E2 -24368.747} C_VEL
LIN {X 0,Y 143.295,Z 557.443,A -85,B 0,C 180,E1 -24372.887,E2 -24372.887} C_VEL
LIN {X 0,Y 143.54,Z 557.416,A -85,B 0,C 180,E1 -24378.706,E2 -24378.706} C_VEL
LIN {X 0,Y 143.627,Z 557.401,A -85,B 0,C 180,E1 -24381.559,E2 -24381.559} C_VEL
LIN {X 0,Y 144.18,Z 557.333,A -85,B 0,C 180,E1 -24390,E2 -24390} C_VEL
LIN {X 0,Y 143.628,Z 557.403,A -85,B 0,C 180,E1 -24398.441,E2 -24398.441} C_VEL
LIN {X 0,Y 143.509,Z 557.417,A -85,B 0,C 180,E1 -24401.63,E2 -24401.63} C_VEL
LIN {X 0,Y 143.305,Z 557.444,A -85,B 0,C 180,E1 -24407.113,E2 -24407.113} C_VEL
LIN {X 0,Y 143.279,Z 557.447,A -85,B 0,C 180,E1 -24411.252,E2 -24411.252} C_VEL
LIN {X 0,Y 143.191,Z 557.455,A -85,B 0,C 180,E1 -24417.934,E2 -24417.934} C_VEL
LIN {X 0,Y 143.17,Z 557.463,A -85,B 0,C 180,E1 -24423.434,E2 -24423.434} C_VEL
LIN {X 0,Y 143.12,Z 557.468,A -85,B 0,C 180,E1 -24429.67,E2 -24429.67} C_VEL
LIN {X 0,Y 143.119,Z 557.468,A -85,B 0,C 180,E1 -24433.43,E2 -24433.43} C_VEL
LIN {X 0,Y 143.087,Z 557.47,A -85,B 0,C 180,E1 -24437.455,E2 -24437.455} C_VEL
LIN {X 0,Y 143.11,Z 557.471,A -85,B 0,C 180,E1 -24441.788,E2 -24441.788} C_VEL
LIN {X 0,Y 143.185,Z 557.459,A -85,B 0,C 180,E1 -24447.321,E2 -24447.321} C_VEL
LIN {X 0,Y 143.19,Z 557.458,A -85,B 0,C 180,E1 -24452.061,E2 -24452.061} C_VEL
LIN {X 0,Y 143.292,Z 557.448,A -85,B 0,C 180,E1 -24458.728,E2 -24458.728} C_VEL
LIN {X 0,Y 143.312,Z 557.44,A -85,B 0,C 180,E1 -24462.887,E2 -24462.887} C_VEL
LIN {X 0,Y 143.593,Z 557.409,A -85,B 0,C 180,E1 -24468.709,E2 -24468.709} C_VEL
LIN {X 0,Y 143.665,Z 557.394,A -85,B 0,C 180,E1 -24471.56,E2 -24471.56} C_VEL
LIN {X 0,Y 144.174,Z 557.333,A -85,B 0,C 180,E1 -24479.999,E2 -24479.999} C_VEL
LIN {X 0,Y 143.656,Z 557.398,A -85,B 0,C 180,E1 -24488.439,E2 -24488.439} C_VEL
LIN {X 0,Y 143.546,Z 557.414,A -85,B 0,C 180,E1 -24491.712,E2 -24491.712} C_VEL
LIN {X 0,Y 143.301,Z 557.441,A -85,B 0,C 180,E1 -24497.112,E2 -24497.112} C_VEL
LIN {X 0,Y 143.272,Z 557.45,A -85,B 0,C 180,E1 -24501.251,E2 -24501.251} C_VEL
LIN {X 0,Y 143.187,Z 557.455,A -85,B 0,C 180,E1 -24507.936,E2 -24507.936} C_VEL
LIN {X 0,Y 143.144,Z 557.464,A -85,B 0,C 180,E1 -24513.422,E2 -24513.422} C_VEL
LIN {X 0,Y 143.058,Z 557.477,A -85,B 0,C 180,E1 -24519.69,E2 -24519.69} C_VEL
LIN {X 0,Y 143.053,Z 557.477,A -85,B 0,C 180,E1 -24523.455,E2 -24523.455} C_VEL
LIN {X 0,Y 143.212,Z 557.458,A -85,B 0,C 180,E1 -24530.361,E2 -24530.361} C_VEL
LIN {X 0,Y 144.096,Z 557.402,A -85,B 0,C 180,E1 -24536.251,E2 -24536.251} C_VEL
LIN {X 0,Y 145.062,Z 561.016,A -85,B 0,C 180,E1 -24538.858,E2 -24538.858} C_VEL
LIN {X 0,Y 145.511,Z 563.706,A -85,B 0,C 180,E1 -24539.317,E2 -24539.317} C_VEL
LIN {X 0,Y 145.394,Z 597.26,A -85,B 0,C 180,E1 -24542.078,E2 -24542.078} C_VEL
LIN {X 0,Y 147.78,Z 650.316,A -85,B 0,C 180,E1 -24546.686,E2 -24546.686} C_VEL
LIN {X 0,Y 147.868,Z 658.479,A -85,B 0,C 180,E1 -24547.652,E2 -24547.652} C_VEL
LIN {X 0,Y 147.117,Z 669.593,A -85,B 0,C 180,E1 -24549.371,E2 -24549.371} C_VEL
LIN {X 0,Y 146.2,Z 679.792,A -85,B 0,C 180,E1 -24551.43,E2 -24551.43} C_VEL
LIN {X 0,Y 145.031,Z 690.349,A -85,B 0,C 180,E1 -24554.182,E2 -24554.182} C_VEL
LIN {X 0,Y 144.27,Z 700.001,A -85,B 0,C 180,E1 -24557.392,E2 -24557.392} C_VEL
LIN {X 0,Y 143.812,Z 708.269,A -85,B 0,C 180,E1 -24560.861,E2 -24560.861} C_VEL
LIN {X 0,Y 144.016,Z 715.014,A -85,B 0,C 180,E1 -24564.399,E2 -24564.399} C_VEL
LIN {X 0,Y 144.501,Z 719.428,A -85,B 0,C 180,E1 -24567.212,E2 -24567.212} C_VEL
LIN {X 0,Y 145.129,Z 723.017,A -85,B 0,C 180,E1 -24570,E2 -24570} C_VEL
LIN {X 0,Y 144.924,Z 724.353,A -85,B 0,C 180,E1 -24571.389,E2 -24571.389} C_VEL
LIN {X 0,Y 143.443,Z 727.145,A -85,B 0,C 180,E1 -24575.623,E2 -24575.623} C_VEL
LIN {X 0,Y 142.729,Z 728.921,A -85,B 0,C 180,E1 -24580.007,E2 -24580.007} C_VEL
LIN {X 0,Y 142.98,Z 729.71,A -85,B 0,C 180,E1 -24584.227,E2 -24584.227} C_VEL
LIN {X 0,Y 143.732,Z 729.776,A -85,B 0,C 180,E1 -24587.06,E2 -24587.06} C_VEL
LIN {X 0,Y 144.978,Z 729.446,A -85,B 0,C 180,E1 -24589.836,E2 -24589.836} C_VEL
LIN {X 0,Y 148.937,Z 727.655,A -85,B 0,C 180,E1 -24595.13,E2 -24595.13} C_VEL
LIN {X 0,Y 151.637,Z 726.185,A -85,B 0,C 180,E1 -24597.611,E2 -24597.611} C_VEL
LIN {X 0,Y 157.008,Z 722.554,A -85,B 0,C 180,E1 -24601.738,E2 -24601.738} C_VEL
LIN {X 0,Y 163.604,Z 717.63,A -85,B 0,C 180,E1 -24605.444,E2 -24605.444} C_VEL
LIN {X 0,Y 171.131,Z 711.13,A -85,B 0,C 180,E1 -24608.776,E2 -24608.776} C_VEL
LIN {X 0,Y 175.684,Z 706.734,A -85,B 0,C 180,E1 -24610.483,E2 -24610.483} C_VEL
LIN {X 0,Y 178.569,Z 703.455,A -85,B 0,C 180,E1 -24611.776,E2 -24611.776} C_VEL
LIN {X 0,Y 182.202,Z 697.906,A -85,B 0,C 180,E1 -24614.124,E2 -24614.124} C_VEL
LIN {X 0,Y 185.989,Z 691.895,A -85,B 0,C 180,E1 -24616.25,E2 -24616.25} C_VEL
LIN {X 0,Y 189.007,Z 687.901,A -85,B 0,C 180,E1 -24617.184,E2 -24617.184} C_VEL
LIN {X 0,Y 197.207,Z 676.64,A -85,B 0,C 180,E1 -24618.836,E2 -24618.836} C_VEL
LIN {X 0,Y 202.999,Z 667.011,A -85,B 0,C 180,E1 -24619.993,E2 -24619.993} C_VEL
LIN {X 0,Y 208.403,Z 656.165,A -85,B 0,C 180,E1 -24621.26,E2 -24621.26} C_VEL
LIN {X 0,Y 212.365,Z 646.168,A -85,B 0,C 180,E1 -24622.583,E2 -24622.583} C_VEL
LIN {X 0,Y 212.714,Z 644.208,A -85,B 0,C 180,E1 -24623.509,E2 -24623.509} C_VEL
LIN {X 0,Y 212.593,Z 643.039,A -85,B 0,C 180,E1 -24625.807,E2 -24625.807} C_VEL
LIN {X 0,Y 211.792,Z 645.145,A -85,B 0,C 180,E1 -24630.149,E2 -24630.149} C_VEL
LIN {X 0,Y 211.568,Z 646.491,A -85,B 0,C 180,E1 -24631.48,E2 -24631.48} C_VEL
LIN {X 0,Y 206.407,Z 656.494,A -85,B 0,C 180,E1 -24632.931,E2 -24632.931} C_VEL
LIN {X 0,Y 199.917,Z 666.458,A -85,B 0,C 180,E1 -24634.743,E2 -24634.743} C_VEL
LIN {X 0,Y 194.065,Z 674.045,A -85,B 0,C 180,E1 -24636.525,E2 -24636.525} C_VEL
LIN {X 0,Y 187.676,Z 680.93,A -85,B 0,C 180,E1 -24638.586,E2 -24638.586} C_VEL
LIN {X 0,Y 181.558,Z 686.46,A -85,B 0,C 180,E1 -24640.791,E2 -24640.791} C_VEL
LIN {X 0,Y 174.392,Z 691.838,A -85,B 0,C 180,E1 -24643.615,E2 -24643.615} C_VEL
LIN {X 0,Y 167.748,Z 695.82,A -85,B 0,C 180,E1 -24646.679,E2 -24646.679} C_VEL
LIN {X 0,Y 161.599,Z 698.542,A -85,B 0,C 180,E1 -24649.983,E2 -24649.983} C_VEL
LIN {X 0,Y 155.511,Z 700.27,A -85,B 0,C 180,E1 -24653.834,E2 -24653.834} C_VEL
LIN {X 0,Y 150.924,Z 700.755,A -85,B 0,C 180,E1 -24657.332,E2 -24657.332} C_VEL
LIN {X 0,Y 147.587,Z 700.509,A -85,B 0,C 180,E1 -24660.339,E2 -24660.339} C_VEL
LIN {X 0,Y 142.863,Z 698.726,A -85,B 0,C 180,E1 -24665.647,E2 -24665.647} C_VEL
LIN {X 0,Y 139.949,Z 696.092,A -85,B 0,C 180,E1 -24670.124,E2 -24670.124} C_VEL
LIN {X 0,Y 137.874,Z 692.297,A -85,B 0,C 180,E1 -24674.767,E2 -24674.767} C_VEL
LIN {X 0,Y 136.631,Z 687.219,A -85,B 0,C 180,E1 -24679.534,E2 -24679.534} C_VEL
LIN {X 0,Y 136.193,Z 680.679,A -85,B 0,C 180,E1 -24684.384,E2 -24684.384} C_VEL
LIN {X 0,Y 136.53,Z 672.928,A -85,B 0,C 180,E1 -24688.947,E2 -24688.947} C_VEL
LIN {X 0,Y 137.394,Z 663.596,A -85,B 0,C 180,E1 -24693.361,E2 -24693.361} C_VEL
LIN {X 0,Y 138.516,Z 654.308,A -85,B 0,C 180,E1 -24696.882,E2 -24696.882} C_VEL
LIN {X 0,Y 139.9,Z 643.124,A -85,B 0,C 180,E1 -24700.301,E2 -24700.301} C_VEL
LIN {X 0,Y 141.425,Z 630.792,A -85,B 0,C 180,E1 -24703.224,E2 -24703.224} C_VEL
LIN {X 0,Y 142.63,Z 619.067,A -85,B 0,C 180,E1 -24705.35,E2 -24705.35} C_VEL
LIN {X 0,Y 143.782,Z 604.807,A -85,B 0,C 180,E1 -24707.227,E2 -24707.227} C_VEL
LIN {X 0,Y 144.562,Z 588.419,A -85,B 0,C 180,E1 -24708.618,E2 -24708.618} C_VEL
LIN {X 0,Y 144.055,Z 585.526,A -85,B 0,C 180,E1 -24708.876,E2 -24708.876} C_VEL
LIN {X 0,Y 136.337,Z 559.148,A -85,B 0,C 180,E1 -24711.671,E2 -24711.671} C_VEL
LIN {X 0,Y 136.151,Z 558.419,A -85,B 0,C 180,E1 -24712.196,E2 -24712.196} C_VEL
LIN {X 0,Y 136.097,Z 558.345,A -85,B 0,C 180,E1 -24715.716,E2 -24715.716} C_VEL
LIN {X 0,Y 136.15,Z 558.336,A -85,B 0,C 180,E1 -24722.318,E2 -24722.318} C_VEL
LIN {X 0,Y 136.246,Z 558.325,A -85,B 0,C 180,E1 -24728.834,E2 -24728.834} C_VEL
LIN {X 0,Y 136.264,Z 558.319,A -85,B 0,C 180,E1 -24735.056,E2 -24735.056} C_VEL
LIN {X 0,Y 136.434,Z 558.302,A -85,B 0,C 180,E1 -24738.168,E2 -24738.168} C_VEL
LIN {X 0,Y 136.553,Z 558.285,A -85,B 0,C 180,E1 -24741.118,E2 -24741.118} C_VEL
LIN {X 0,Y 137.137,Z 558.21,A -85,B 0,C 180,E1 -24750,E2 -24750} C_VEL
LIN {X 0,Y 136.554,Z 558.283,A -85,B 0,C 180,E1 -24758.882,E2 -24758.882} C_VEL
LIN {X 0,Y 136.444,Z 558.298,A -85,B 0,C 180,E1 -24761.89,E2 -24761.89} C_VEL
LIN {X 0,Y 136.245,Z 558.321,A -85,B 0,C 180,E1 -24768.029,E2 -24768.029} C_VEL
LIN {X 0,Y 136.199,Z 558.33,A -85,B 0,C 180,E1 -24771.746,E2 -24771.746} C_VEL
LIN {X 0,Y 136.101,Z 558.339,A -85,B 0,C 180,E1 -24778.614,E2 -24778.614} C_VEL
LIN {X 0,Y 136.084,Z 558.343,A -85,B 0,C 180,E1 -24784.616,E2 -24784.616} C_VEL
LIN {X 0,Y 136.088,Z 558.343,A -85,B 0,C 180,E1 -24789.225,E2 -24789.225} C_VEL
LIN {X 0,Y 136.055,Z 558.349,A -85,B 0,C 180,E1 -24793.681,E2 -24793.681} C_VEL
LIN {X 0,Y 136.048,Z 558.347,A -85,B 0,C 180,E1 -24797.811,E2 -24797.811} C_VEL
LIN {X 0,Y 136.06,Z 558.349,A -85,B 0,C 180,E1 -24801.694,E2 -24801.694} C_VEL
LIN {X 0,Y 136.09,Z 558.339,A -85,B 0,C 180,E1 -24805.716,E2 -24805.716} C_VEL
LIN {X 0,Y 136.146,Z 558.334,A -85,B 0,C 180,E1 -24812.315,E2 -24812.315} C_VEL
LIN {X 0,Y 136.26,Z 558.324,A -85,B 0,C 180,E1 -24818.834,E2 -24818.834} C_VEL
LIN {X 0,Y 136.276,Z 558.321,A -85,B 0,C 180,E1 -24825.056,E2 -24825.056} C_VEL
LIN {X 0,Y 136.496,Z 558.295,A -85,B 0,C 180,E1 -24828.113,E2 -24828.113} C_VEL
LIN {X 0,Y 136.592,Z 558.275,A -85,B 0,C 180,E1 -24831.119,E2 -24831.119} C_VEL
LIN {X 0,Y 137.131,Z 558.21,A -85,B 0,C 180,E1 -24839.999,E2 -24839.999} C_VEL
LIN {X 0,Y 136.585,Z 558.277,A -85,B 0,C 180,E1 -24848.879,E2 -24848.879} C_VEL
LIN {X 0,Y 136.489,Z 558.294,A -85,B 0,C 180,E1 -24851.954,E2 -24851.954} C_VEL
LIN {X 0,Y 136.24,Z 558.32,A -85,B 0,C 180,E1 -24858.029,E2 -24858.029} C_VEL
LIN {X 0,Y 136.193,Z 558.331,A -85,B 0,C 180,E1 -24861.745,E2 -24861.745} C_VEL
LIN {X 0,Y 136.114,Z 558.338,A -85,B 0,C 180,E1 -24868.628,E2 -24868.628} C_VEL
LIN {X 0,Y 136.041,Z 558.347,A -85,B 0,C 180,E1 -24874.628,E2 -24874.628} C_VEL
LIN {X 0,Y 136.028,Z 558.353,A -85,B 0,C 180,E1 -24879.198,E2 -24879.198} C_VEL
LIN {X 0,Y 135.995,Z 558.356,A -85,B 0,C 180,E1 -24883.657,E2 -24883.657} C_VEL
LIN {X 0,Y 136.206,Z 558.332,A -85,B 0,C 180,E1 -24890.711,E2 -24890.711} C_VEL
LIN {X 0,Y 137.263,Z 558.344,A -85,B 0,C 180,E1 -24897.153,E2 -24897.153} C_VEL
LIN {X 0,Y 137.666,Z 560.123,A -85,B 0,C 180,E1 -24898.258,E2 -24898.258} C_VEL
LIN {X 0,Y 138.605,Z 565.584,A -85,B 0,C 180,E1 -24898.899,E2 -24898.899} C_VEL
LIN {X 0,Y 138.302,Z 590.094,A -85,B 0,C 180,E1 -24901.031,E2 -24901.031} C_VEL
LIN {X 0,Y 139.889,Z 635.251,A -85,B 0,C 180,E1 -24905.1,E2 -24905.1} C_VEL
LIN {X 0,Y 140.749,Z 652.375,A -85,B 0,C 180,E1 -24906.797,E2 -24906.797} C_VEL
LIN {X 0,Y 140.762,Z 658.545,A -85,B 0,C 180,E1 -24907.623,E2 -24907.623} C_VEL
LIN {X 0,Y 140.019,Z 669.41,A -85,B 0,C 180,E1 -24909.43,E2 -24909.43} C_VEL
LIN {X 0,Y 139.108,Z 679.361,A -85,B 0,C 180,E1 -24911.593,E2 -24911.593} C_VEL
LIN {X 0,Y 137.964,Z 689.794,A -85,B 0,C 180,E1 -24914.488,E2 -24914.488} C_VEL
LIN {X 0,Y 137.223,Z 700.119,A -85,B 0,C 180,E1 -24918.179,E2 -24918.179} C_VEL
LIN {X 0,Y 136.956,Z 708.238,A -85,B 0,C 180,E1 -24921.887,E2 -24921.887} C_VEL
LIN {X 0,Y 137.3,Z 714.753,A -85,B 0,C 180,E1 -24925.596,E2 -24925.596} C_VEL
LIN {X 0,Y 138.227,Z 720.752,A -85,B 0,C 180,E1 -24930,E2 -24930} C_VEL
LIN {X 0,Y 138.147,Z 722.231,A -85,B 0,C 180,E1 -24931.457,E2 -24931.457} C_VEL
LIN {X 0,Y 136.572,Z 725.24,A -85,B 0,C 180,E1 -24935.907,E2 -24935.907} C_VEL
LIN {X 0,Y 135.862,Z 727.267,A -85,B 0,C 180,E1 -24940.631,E2 -24940.631} C_VEL
LIN {X 0,Y 136.169,Z 728.23,A -85,B 0,C 180,E1 -24944.954,E2 -24944.954} C_VEL
LIN {X 0,Y 138.383,Z 728.276,A -85,B 0,C 180,E1 -24950.824,E2 -24950.824} C_VEL
LIN {X 0,Y 140.278,Z 727.764,A -85,B 0,C 180,E1 -24953.628,E2 -24953.628} C_VEL
LIN {X 0,Y 142.558,Z 726.843,A -85,B 0,C 180,E1 -24956.339,E2 -24956.339} C_VEL
LIN {X 0,Y 145.397,Z 725.543,A -85,B 0,C 180,E1 -24958.905,E2 -24958.905} C_VEL
LIN {X 0,Y 150.543,Z 722.604,A -85,B 0,C 180,E1 -24962.828,E2 -24962.828} C_VEL
LIN {X 0,Y 157.883,Z 717.79,A -85,B 0,C 180,E1 -24966.936,E2 -24966.936} C_VEL
LIN {X 0,Y 164.513,Z 712.733,A -85,B 0,C 180,E1 -24969.85,E2 -24969.85} C_VEL
LIN {X 0,Y 172.485,Z 705.8,A -85,B 0,C 180,E1 -24972.742,E2 -24972.742} C_VEL
LIN {X 0,Y 179.461,Z 698.873,A -85,B 0,C 180,E1 -24974.821,E2 -24974.821} C_VEL
LIN {X 0,Y 187.692,Z 689.495,A -85,B 0,C 180,E1 -24976.899,E2 -24976.899} C_VEL
LIN {X 0,Y 189.007,Z 687.901,A -85,B 0,C 180,E1 -24977.184,E2 -24977.184} C_VEL
LIN {X 0,Y 192.103,Z 683.774,A -85,B 0,C 180,E1 -24978.056,E2 -24978.056} C_VEL
LIN {X 0,Y 196.206,Z 676.974,A -85,B 0,C 180,E1 -24979.809,E2 -24979.809} C_VEL
LIN {X 0,Y 199.979,Z 669.806,A -85,B 0,C 180,E1 -24981.475,E2 -24981.475} C_VEL
LIN {X 0,Y 202.492,Z 665.098,A -85,B 0,C 180,E1 -24982.214,E2 -24982.214} C_VEL
LIN {X 0,Y 207.204,Z 655.97,A -85,B 0,C 180,E1 -24983.314,E2 -24983.314} C_VEL
LIN {X 0,Y 208.953,Z 652.128,A -85,B 0,C 180,E1 -24983.823,E2 -24983.823} C_VEL
LIN {X 0,Y 209.691,Z 650.188,A -85,B 0,C 180,E1 -24984.508,E2 -24984.508} C_VEL
LIN {X 0,Y 209.651,Z 649.806,A -85,B 0,C 180,E1 -24985.259,E2 -24985.259} C_VEL
LIN {X 0,Y 209.05,Z 650.159,A -85,B 0,C 180,E1 -24987.46,E2 -24987.46} C_VEL
LIN {X 0,Y 208.584,Z 651.259,A -85,B 0,C 180,E1 -24989.642,E2 -24989.642} C_VEL
LIN {X 0,Y 208.293,Z 651.878,A -85,B 0,C 180,E1 -24990.16,E2 -24990.16} C_VEL
LIN {X 0,Y 202.204,Z 662.179,A -85,B 0,C 180,E1 -24991.713,E2 -24991.713} C_VEL
LIN {X 0,Y 195.944,Z 670.748,A -85,B 0,C 180,E1 -24993.362,E2 -24993.362} C_VEL
LIN {X 0,Y 189.178,Z 678.432,A -85,B 0,C 180,E1 -24995.296,E2 -24995.296} C_VEL
LIN {X 0,Y 181.244,Z 685.855,A -85,B 0,C 180,E1 -24997.787,E2 -24997.787} C_VEL
LIN {X 0,Y 174.913,Z 690.748,A -85,B 0,C 180,E1 -25000.031,E2 -25000.031} C_VEL
LIN {X 0,Y 167.553,Z 695.364,A -85,B 0,C 180,E1 -25002.926,E2 -25002.926} C_VEL
LIN {X 0,Y 162.904,Z 697.707,A -85,B 0,C 180,E1 -25004.999,E2 -25004.999} C_VEL
LIN {X 0,Y 158.522,Z 699.538,A -85,B 0,C 180,E1 -25007.194,E2 -25007.194} C_VEL
LIN {X 0,Y 153.244,Z 701.07,A -85,B 0,C 180,E1 -25010.161,E2 -25010.161} C_VEL
LIN {X 0,Y 146.782,Z 702.041,A -85,B 0,C 180,E1 -25014.506,E2 -25014.506} C_VEL
LIN {X 0,Y 143.418,Z 701.926,A -85,B 0,C 180,E1 -25017.192,E2 -25017.192} C_VEL
LIN {X 0,Y 140.354,Z 701.376,A -85,B 0,C 180,E1 -25020.001,E2 -25020.001} C_VEL
LIN {X 0,Y 137.653,Z 700.313,A -85,B 0,C 180,E1 -25022.928,E2 -25022.928} C_VEL
LIN {X 0,Y 134.532,Z 698.18,A -85,B 0,C 180,E1 -25027.004,E2 -25027.004} C_VEL
LIN {X 0,Y 131.648,Z 694.253,A -85,B 0,C 180,E1 -25032.331,E2 -25032.331} C_VEL
LIN {X 0,Y 129.981,Z 689.419,A -85,B 0,C 180,E1 -25037.302,E2 -25037.302} C_VEL
LIN {X 0,Y 129.174,Z 683.139,A -85,B 0,C 180,E1 -25042.388,E2 -25042.388} C_VEL
LIN {X 0,Y 129.275,Z 675.255,A -85,B 0,C 180,E1 -25047.524,E2 -25047.524} C_VEL
LIN {X 0,Y 129.976,Z 666.818,A -85,B 0,C 180,E1 -25051.889,E2 -25051.889} C_VEL
LIN {X 0,Y 131.116,Z 656.645,A -85,B 0,C 180,E1 -25056.131,E2 -25056.131} C_VEL
LIN {X 0,Y 132.621,Z 644.868,A -85,B 0,C 180,E1 -25059.983,E2 -25059.983} C_VEL
LIN {X 0,Y 134.08,Z 633.208,A -85,B 0,C 180,E1 -25062.956,E2 -25062.956} C_VEL
LIN {X 0,Y 135.35,Z 621.407,A -85,B 0,C 180,E1 -25065.295,E2 -25065.295} C_VEL
LIN {X 0,Y 136.488,Z 608.335,A -85,B 0,C 180,E1 -25067.203,E2 -25067.203} C_VEL
LIN {X 0,Y 137.328,Z 594.856,A -85,B 0,C 180,E1 -25068.549,E2 -25068.549} C_VEL
LIN {X 0,Y 137.454,Z 588.046,A -85,B 0,C 180,E1 -25069.108,E2 -25069.108} C_VEL
LIN {X 0,Y 129.257,Z 560.117,A -85,B 0,C 180,E1 -25072.166,E2 -25072.166} C_VEL
LIN {X 0,Y 129.098,Z 559.303,A -85,B 0,C 180,E1 -25072.727,E2 -25072.727} C_VEL
LIN {X 0,Y 129.002,Z 559.229,A -85,B 0,C 180,E1 -25076.99,E2 -25076.99} C_VEL
LIN {X 0,Y 129.053,Z 559.222,A -85,B 0,C 180,E1 -25080.652,E2 -25080.652} C_VEL
LIN {X 0,Y 129.11,Z 559.215,A -85,B 0,C 180,E1 -25087.729,E2 -25087.729} C_VEL
LIN {X 0,Y 129.152,Z 559.208,A -85,B 0,C 180,E1 -25090.944,E2 -25090.944} C_VEL
LIN {X 0,Y 129.379,Z 559.182,A -85,B 0,C 180,E1 -25097.905,E2 -25097.905} C_VEL
LIN {X 0,Y 129.476,Z 559.166,A -85,B 0,C 180,E1 -25100.629,E2 -25100.629} C_VEL
LIN {X 0,Y 130.092,Z 559.087,A -85,B 0,C 180,E1 -25110,E2 -25110} C_VEL
LIN {X 0,Y 129.477,Z 559.164,A -85,B 0,C 180,E1 -25119.372,E2 -25119.372} C_VEL
LIN {X 0,Y 129.348,Z 559.183,A -85,B 0,C 180,E1 -25122.553,E2 -25122.553} C_VEL
LIN {X 0,Y 129.155,Z 559.202,A -85,B 0,C 180,E1 -25129.056,E2 -25129.056} C_VEL
LIN {X 0,Y 129.111,Z 559.215,A -85,B 0,C 180,E1 -25132.398,E2 -25132.398} C_VEL
LIN {X 0,Y 129.03,Z 559.223,A -85,B 0,C 180,E1 -25135.832,E2 -25135.832} C_VEL
LIN {X 0,Y 129.019,Z 559.221,A -85,B 0,C 180,E1 -25139.357,E2 -25139.357} C_VEL
LIN {X 0,Y 129.026,Z 559.222,A -85,B 0,C 180,E1 -25145.208,E2 -25145.208} C_VEL
LIN {X 0,Y 129.007,Z 559.227,A -85,B 0,C 180,E1 -25150.823,E2 -25150.823} C_VEL
LIN {X 0,Y 128.977,Z 559.225,A -85,B 0,C 180,E1 -25155.102,E2 -25155.102} C_VEL
LIN {X 0,Y 128.986,Z 559.23,A -85,B 0,C 180,E1 -25159.711,E2 -25159.711} C_VEL
LIN {X 0,Y 128.993,Z 559.222,A -85,B 0,C 180,E1 -25164.809,E2 -25164.809} C_VEL
LIN {X 0,Y 129.034,Z 559.223,A -85,B 0,C 180,E1 -25170.645,E2 -25170.645} C_VEL
LIN {X 0,Y 129.111,Z 559.214,A -85,B 0,C 180,E1 -25177.601,E2 -25177.601} C_VEL
LIN {X 0,Y 129.166,Z 559.203,A -85,B 0,C 180,E1 -25180.944,E2 -25180.944} C_VEL
LIN {X 0,Y 129.415,Z 559.177,A -85,B 0,C 180,E1 -25187.819,E2 -25187.819} C_VEL
LIN {X 0,Y 129.517,Z 559.157,A -85,B 0,C 180,E1 -25190.63,E2 -25190.63} C_VEL
LIN {X 0,Y 130.086,Z 559.087,A -85,B 0,C 180,E1 -25199.999,E2 -25199.999} C_VEL
LIN {X 0,Y 129.511,Z 559.157,A -85,B 0,C 180,E1 -25209.368,E2 -25209.368} C_VEL
LIN {X 0,Y 129.391,Z 559.18,A -85,B 0,C 180,E1 -25212.547,E2 -25212.547} C_VEL
LIN {X 0,Y 129.15,Z 559.205,A -85,B 0,C 180,E1 -25219.056,E2 -25219.056} C_VEL
LIN {X 0,Y 129.105,Z 559.216,A -85,B 0,C 180,E1 -25222.398,E2 -25222.398} C_VEL
LIN {X 0,Y 129.033,Z 559.223,A -85,B 0,C 180,E1 -25229.373,E2 -25229.373} C_VEL
LIN {X 0,Y 128.957,Z 559.227,A -85,B 0,C 180,E1 -25235.168,E2 -25235.168} C_VEL
LIN {X 0,Y 128.931,Z 559.238,A -85,B 0,C 180,E1 -25240.851,E2 -25240.851} C_VEL
LIN {X 0,Y 128.922,Z 559.239,A -85,B 0,C 180,E1 -25245.126,E2 -25245.126} C_VEL
LIN {X 0,Y 129.08,Z 559.218,A -85,B 0,C 180,E1 -25249.662,E2 -25249.662} C_VEL
LIN {X 0,Y 130.242,Z 559.311,A -85,B 0,C 180,E1 -25257.229,E2 -25257.229} C_VEL
LIN {X 0,Y 130.479,Z 560.332,A -85,B 0,C 180,E1 -25257.678,E2 -25257.678} C_VEL
LIN {X 0,Y 131.614,Z 566.45,A -85,B 0,C 180,E1 -25258.379,E2 -25258.379} C_VEL
LIN {X 0,Y 131.355,Z 592.448,A -85,B 0,C 180,E1 -25260.767,E2 -25260.767} C_VEL
LIN {X 0,Y 132.835,Z 635.773,A -85,B 0,C 180,E1 -25264.896,E2 -25264.896} C_VEL
LIN {X 0,Y 133.633,Z 651.458,A -85,B 0,C 180,E1 -25266.564,E2 -25266.564} C_VEL
LIN {X 0,Y 133.652,Z 658.6,A -85,B 0,C 180,E1 -25267.59,E2 -25267.59} C_VEL
LIN {X 0,Y 132.928,Z 669.17,A -85,B 0,C 180,E1 -25269.497,E2 -25269.497} C_VEL
LIN {X 0,Y 131.889,Z 680.39,A -85,B 0,C 180,E1 -25272.158,E2 -25272.158} C_VEL
LIN {X 0,Y 130.829,Z 690.294,A -85,B 0,C 180,E1 -25275.223,E2 -25275.223} C_VEL
LIN {X 0,Y 130.24,Z 700.21,A -85,B 0,C 180,E1 -25279.113,E2 -25279.113} C_VEL
LIN {X 0,Y 130.139,Z 708.031,A -85,B 0,C 180,E1 -25283.021,E2 -25283.021} C_VEL
LIN {X 0,Y 130.604,Z 714.323,A -85,B 0,C 180,E1 -25286.915,E2 -25286.915} C_VEL
LIN {X 0,Y 131.322,Z 718.374,A -85,B 0,C 180,E1 -25290,E2 -25290} C_VEL
LIN {X 0,Y 131.396,Z 719.993,A -85,B 0,C 180,E1 -25291.532,E2 -25291.532} C_VEL
LIN {X 0,Y 129.732,Z 723.229,A -85,B 0,C 180,E1 -25296.22,E2 -25296.22} C_VEL
LIN {X 0,Y 129.031,Z 725.521,A -85,B 0,C 180,E1 -25301.362,E2 -25301.362} C_VEL
LIN {X 0,Y 129.419,Z 726.649,A -85,B 0,C 180,E1 -25305.754,E2 -25305.754} C_VEL
LIN {X 0,Y 131.83,Z 727.043,A -85,B 0,C 180,E1 -25311.911,E2 -25311.911} C_VEL
LIN {X 0,Y 136.267,Z 725.937,A -85,B 0,C 180,E1 -25317.656,E2 -25317.656} C_VEL
LIN {X 0,Y 139.239,Z 724.853,A -85,B 0,C 180,E1 -25320.313,E2 -25320.313} C_VEL
LIN {X 0,Y 143.997,Z 722.573,A -85,B 0,C 180,E1 -25323.933,E2 -25323.933} C_VEL
LIN {X 0,Y 150.155,Z 719.155,A -85,B 0,C 180,E1 -25327.477,E2 -25327.477} C_VEL
LIN {X 0,Y 156.795,Z 714.906,A -85,B 0,C 180,E1 -25330.535,E2 -25330.535} C_VEL
LIN {X 0,Y 164.609,Z 709.095,A -85,B 0,C 180,E1 -25333.464,E2 -25333.464} C_VEL
LIN {X 0,Y 173.177,Z 701.673,A -85,B 0,C 180,E1 -25336.113,E2 -25336.113} C_VEL
LIN {X 0,Y 181.527,Z 693.393,A -85,B 0,C 180,E1 -25338.182,E2 -25338.182} C_VEL
LIN {X 0,Y 188.884,Z 684.875,A -85,B 0,C 180,E1 -25339.707,E2 -25339.707} C_VEL
LIN {X 0,Y 197.255,Z 673.625,A -85,B 0,C 180,E1 -25341.202,E2 -25341.202} C_VEL
LIN {X 0,Y 202.492,Z 665.098,A -85,B 0,C 180,E1 -25342.214,E2 -25342.214} C_VEL
LIN {X 0,Y 203.319,Z 663.311,A -85,B 0,C 180,E1 -25342.699,E2 -25342.699} C_VEL
LIN {X 0,Y 204.305,Z 660.015,A -85,B 0,C 180,E1 -25344.72,E2 -25344.72} C_VEL
LIN {X 0,Y 204.963,Z 658.654,A -85,B 0,C 180,E1 -25345.042,E2 -25345.042} C_VEL
LIN {X 0,Y 205.488,Z 657.662,A -85,B 0,C 180,E1 -25345.167,E2 -25345.167} C_VEL
LIN {X 0,Y 206.17,Z 656.141,A -85,B 0,C 180,E1 -25345.714,E2 -25345.714} C_VEL
LIN {X 0,Y 205.814,Z 656.231,A -85,B 0,C 180,E1 -25346.883,E2 -25346.883} C_VEL
LIN {X 0,Y 205.355,Z 656.836,A -85,B 0,C 180,E1 -25348.285,E2 -25348.285} C_VEL
LIN {X 0,Y 204.311,Z 658.528,A -85,B 0,C 180,E1 -25348.938,E2 -25348.938} C_VEL
LIN {X 0,Y 198.588,Z 666.916,A -85,B 0,C 180,E1 -25350.301,E2 -25350.301} C_VEL
LIN {X 0,Y 191.297,Z 675.711,A -85,B 0,C 180,E1 -25352.128,E2 -25352.128} C_VEL
LIN {X 0,Y 184.364,Z 682.699,A -85,B 0,C 180,E1 -25354,E2 -25354} C_VEL
LIN {X 0,Y 176.168,Z 689.425,A -85,B 0,C 180,E1 -25356.489,E2 -25356.489} C_VEL
LIN {X 0,Y 168.186,Z 694.707,A -85,B 0,C 180,E1 -25359.196,E2 -25359.196} C_VEL
LIN {X 0,Y 160.637,Z 698.634,A -85,B 0,C 180,E1 -25362.167,E2 -25362.167} C_VEL
LIN {X 0,Y 155.894,Z 700.513,A -85,B 0,C 180,E1 -25364.307,E2 -25364.307} C_VEL
LIN {X 0,Y 151.358,Z 701.933,A -85,B 0,C 180,E1 -25366.576,E2 -25366.576} C_VEL
LIN {X 0,Y 147.065,Z 702.848,A -85,B 0,C 180,E1 -25368.981,E2 -25368.981} C_VEL
LIN {X 0,Y 141.815,Z 703.358,A -85,B 0,C 180,E1 -25372.359,E2 -25372.359} C_VEL
LIN {X 0,Y 135.852,Z 702.816,A -85,B 0,C 180,E1 -25377.036,E2 -25377.036} C_VEL
LIN {X 0,Y 132.771,Z 701.893,A -85,B 0,C 180,E1 -25380.001,E2 -25380.001} C_VEL
LIN {X 0,Y 130.02,Z 700.452,A -85,B 0,C 180,E1 -25383.1,E2 -25383.1} C_VEL
LIN {X 0,Y 126.577,Z 697.377,A -85,B 0,C 180,E1 -25388.017,E2 -25388.017} C_VEL
LIN {X 0,Y 124.117,Z 693.208,A -85,B 0,C 180,E1 -25393.092,E2 -25393.092} C_VEL
LIN {X 0,Y 122.611,Z 687.701,A -85,B 0,C 180,E1 -25398.378,E2 -25398.378} C_VEL
LIN {X 0,Y 122.051,Z 680.65,A -85,B 0,C 180,E1 -25403.772,E2 -25403.772} C_VEL
LIN {X 0,Y 122.293,Z 673.411,A -85,B 0,C 180,E1 -25408.303,E2 -25408.303} C_VEL
LIN {X 0,Y 123.071,Z 664.476,A -85,B 0,C 180,E1 -25412.855,E2 -25412.855} C_VEL
LIN {X 0,Y 124.351,Z 654.023,A -85,B 0,C 180,E1 -25417.152,E2 -25417.152} C_VEL
LIN {X 0,Y 125.673,Z 643.518,A -85,B 0,C 180,E1 -25420.551,E2 -25420.551} C_VEL
LIN {X 0,Y 127.223,Z 631.242,A -85,B 0,C 180,E1 -25423.678,E2 -25423.678} C_VEL
LIN {X 0,Y 128.595,Z 618.497,A -85,B 0,C 180,E1 -25426.116,E2 -25426.116} C_VEL
LIN {X 0,Y 129.656,Z 605.075,A -85,B 0,C 180,E1 -25427.965,E2 -25427.965} C_VEL
LIN {X 0,Y 130.502,Z 589.443,A -85,B 0,C 180,E1 -25429.413,E2 -25429.413} C_VEL
LIN {X 0,Y 122.159,Z 560.866,A -85,B 0,C 180,E1 -25432.774,E2 -25432.774} C_VEL
LIN {X 0,Y 122.025,Z 560.139,A -85,B 0,C 180,E1 -25433.524,E2 -25433.524} C_VEL
LIN {X 0,Y 121.945,Z 560.108,A -85,B 0,C 180,E1 -25439.827,E2 -25439.827} C_VEL
LIN {X 0,Y 121.986,Z 560.099,A -85,B 0,C 180,E1 -25446.217,E2 -25446.217} C_VEL
LIN {X 0,Y 122.046,Z 560.095,A -85,B 0,C 180,E1 -25449.788,E2 -25449.788} C_VEL
LIN {X 0,Y 122.241,Z 560.069,A -85,B 0,C 180,E1 -25456.705,E2 -25456.705} C_VEL
LIN {X 0,Y 122.409,Z 560.047,A -85,B 0,C 180,E1 -25460.082,E2 -25460.082} C_VEL
LIN {X 0,Y 122.599,Z 560.025,A -85,B 0,C 180,E1 -25466.714,E2 -25466.714} C_VEL
LIN {X 0,Y 123.045,Z 559.965,A -85,B 0,C 180,E1 -25470,E2 -25470} C_VEL
LIN {X 0,Y 122.426,Z 560.047,A -85,B 0,C 180,E1 -25476.593,E2 -25476.593} C_VEL
LIN {X 0,Y 122.413,Z 560.042,A -85,B 0,C 180,E1 -25479.918,E2 -25479.918} C_VEL
LIN {X 0,Y 122.243,Z 560.069,A -85,B 0,C 180,E1 -25483.295,E2 -25483.295} C_VEL
LIN {X 0,Y 122.048,Z 560.089,A -85,B 0,C 180,E1 -25490.212,E2 -25490.212} C_VEL
LIN {X 0,Y 121.985,Z 560.103,A -85,B 0,C 180,E1 -25493.784,E2 -25493.784} C_VEL
LIN {X 0,Y 121.932,Z 560.107,A -85,B 0,C 180,E1 -25500.162,E2 -25500.162} C_VEL
LIN {X 0,Y 121.938,Z 560.101,A -85,B 0,C 180,E1 -25506.204,E2 -25506.204} C_VEL
LIN {X 0,Y 121.932,Z 560.109,A -85,B 0,C 180,E1 -25511.468,E2 -25511.468} C_VEL
LIN {X 0,Y 121.914,Z 560.111,A -85,B 0,C 180,E1 -25518.539,E2 -25518.539} C_VEL
LIN {X 0,Y 121.946,Z 560.1,A -85,B 0,C 180,E1 -25524.806,E2 -25524.806} C_VEL
LIN {X 0,Y 121.942,Z 560.108,A -85,B 0,C 180,E1 -25529.825,E2 -25529.825} C_VEL
LIN {X 0,Y 121.986,Z 560.1,A -85,B 0,C 180,E1 -25536.214,E2 -25536.214} C_VEL
LIN {X 0,Y 122.057,Z 560.093,A -85,B 0,C 180,E1 -25539.788,E2 -25539.788} C_VEL
LIN {X 0,Y 122.362,Z 560.055,A -85,B 0,C 180,E1 -25547.525,E2 -25547.525} C_VEL
LIN {X 0,Y 122.446,Z 560.04,A -85,B 0,C 180,E1 -25550.084,E2 -25550.084} C_VEL
LIN {X 0,Y 122.605,Z 560.025,A -85,B 0,C 180,E1 -25556.713,E2 -25556.713} C_VEL
LIN {X 0,Y 123.04,Z 559.964,A -85,B 0,C 180,E1 -25559.999,E2 -25559.999} C_VEL
LIN {X 0,Y 122.441,Z 560.044,A -85,B 0,C 180,E1 -25566.591,E2 -25566.591} C_VEL
LIN {X 0,Y 122.442,Z 560.038,A -85,B 0,C 180,E1 -25569.914,E2 -25569.914} C_VEL
LIN {X 0,Y 122.26,Z 560.068,A -85,B 0,C 180,E1 -25573.292,E2 -25573.292} C_VEL
LIN {X 0,Y 122.042,Z 560.092,A -85,B 0,C 180,E1 -25580.212,E2 -25580.212} C_VEL
LIN {X 0,Y 121.98,Z 560.102,A -85,B 0,C 180,E1 -25583.784,E2 -25583.784} C_VEL
LIN {X 0,Y 121.937,Z 560.107,A -85,B 0,C 180,E1 -25590.171,E2 -25590.171} C_VEL
LIN {X 0,Y 121.881,Z 560.107,A -85,B 0,C 180,E1 -25596.171,E2 -25596.171} C_VEL
LIN {X 0,Y 121.87,Z 560.116,A -85,B 0,C 180,E1 -25601.438,E2 -25601.438} C_VEL
LIN {X 0,Y 121.957,Z 560.107,A -85,B 0,C 180,E1 -25608.515,E2 -25608.515} C_VEL
LIN {X 0,Y 122.974,Z 560.097,A -85,B 0,C 180,E1 -25616.487,E2 -25616.487} C_VEL
LIN {X 0,Y 123.258,Z 560.983,A -85,B 0,C 180,E1 -25617.054,E2 -25617.054} C_VEL
LIN {X 0,Y 124.617,Z 566.51,A -85,B 0,C 180,E1 -25617.772,E2 -25617.772} C_VEL
LIN {X 0,Y 124.37,Z 599.304,A -85,B 0,C 180,E1 -25621.005,E2 -25621.005} C_VEL
LIN {X 0,Y 126.264,Z 647.146,A -85,B 0,C 180,E1 -25625.928,E2 -25625.928} C_VEL
LIN {X 0,Y 126.665,Z 657.063,A -85,B 0,C 180,E1 -25627.361,E2 -25627.361} C_VEL
LIN {X 0,Y 125.866,Z 668.583,A -85,B 0,C 180,E1 -25629.575,E2 -25629.575} C_VEL
LIN {X 0,Y 124.847,Z 679.626,A -85,B 0,C 180,E1 -25632.388,E2 -25632.388} C_VEL
LIN {X 0,Y 123.838,Z 689.407,A -85,B 0,C 180,E1 -25635.618,E2 -25635.618} C_VEL
LIN {X 0,Y 123.36,Z 698.432,A -85,B 0,C 180,E1 -25639.33,E2 -25639.33} C_VEL
LIN {X 0,Y 123.299,Z 706.36,A -85,B 0,C 180,E1 -25643.454,E2 -25643.454} C_VEL
LIN {X 0,Y 123.835,Z 712.741,A -85,B 0,C 180,E1 -25647.56,E2 -25647.56} C_VEL
LIN {X 0,Y 124.411,Z 715.929,A -85,B 0,C 180,E1 -25650,E2 -25650} C_VEL
LIN {X 0,Y 124.629,Z 717.7,A -85,B 0,C 180,E1 -25651.615,E2 -25651.615} C_VEL
LIN {X 0,Y 122.932,Z 721.119,A -85,B 0,C 180,E1 -25656.565,E2 -25656.565} C_VEL
LIN {X 0,Y 122.281,Z 724.111,A -85,B 0,C 180,E1 -25663.29,E2 -25663.29} C_VEL
LIN {X 0,Y 122.707,Z 724.994,A -85,B 0,C 180,E1 -25666.64,E2 -25666.64} C_VEL
LIN {X 0,Y 123.743,Z 725.525,A -85,B 0,C 180,E1 -25669.923,E2 -25669.923} C_VEL
LIN {X 0,Y 127.464,Z 725.511,A -85,B 0,C 180,E1 -25676.173,E2 -25676.173} C_VEL
LIN {X 0,Y 130.074,Z 724.979,A -85,B 0,C 180,E1 -25679.095,E2 -25679.095} C_VEL
LIN {X 0,Y 133.173,Z 724.07,A -85,B 0,C 180,E1 -25681.851,E2 -25681.851} C_VEL
LIN {X 0,Y 137.391,Z 722.401,A -85,B 0,C 180,E1 -25685.071,E2 -25685.071} C_VEL
LIN {X 0,Y 144.587,Z 719.052,A -85,B 0,C 180,E1 -25689.189,E2 -25689.189} C_VEL
LIN {X 0,Y 151.483,Z 715.161,A -85,B 0,C 180,E1 -25692.276,E2 -25692.276} C_VEL
LIN {X 0,Y 161.558,Z 708.361,A -85,B 0,C 180,E1 -25695.867,E2 -25695.867} C_VEL
LIN {X 0,Y 169.703,Z 701.88,A -85,B 0,C 180,E1 -25698.195,E2 -25698.195} C_VEL
LIN {X 0,Y 179.866,Z 692.426,A -85,B 0,C 180,E1 -25700.505,E2 -25700.505} C_VEL
LIN {X 0,Y 187.506,Z 684.133,A -85,B 0,C 180,E1 -25701.914,E2 -25701.914} C_VEL
LIN {X 0,Y 196.046,Z 673.055,A -85,B 0,C 180,E1 -25703.331,E2 -25703.331} C_VEL
LIN {X 0,Y 203.117,Z 661.931,A -85,B 0,C 180,E1 -25704.632,E2 -25704.632} C_VEL
LIN {X 0,Y 204.963,Z 658.654,A -85,B 0,C 180,E1 -25705.042,E2 -25705.042} C_VEL
LIN {X 0,Y 205.236,Z 658.002,A -85,B 0,C 180,E1 -25705.355,E2 -25705.355} C_VEL
LIN {X 0,Y 204.822,Z 658.332,A -85,B 0,C 180,E1 -25706.053,E2 -25706.053} C_VEL
LIN {X 0,Y 203.174,Z 660.633,A -85,B 0,C 180,E1 -25707.059,E2 -25707.059} C_VEL
LIN {X 0,Y 201.526,Z 662.951,A -85,B 0,C 180,E1 -25707.652,E2 -25707.652} C_VEL
LIN {X 0,Y 198.54,Z 667.111,A -85,B 0,C 180,E1 -25708.345,E2 -25708.345} C_VEL
LIN {X 0,Y 191.921,Z 675.168,A -85,B 0,C 180,E1 -25709.615,E2 -25709.615} C_VEL
LIN {X 0,Y 188.533,Z 678.737,A -85,B 0,C 180,E1 -25710.372,E2 -25710.372} C_VEL
LIN {X 0,Y 179.601,Z 686.741,A -85,B 0,C 180,E1 -25712.627,E2 -25712.627} C_VEL
LIN {X 0,Y 171.631,Z 692.592,A -85,B 0,C 180,E1 -25714.95,E2 -25714.95} C_VEL
LIN {X 0,Y 164.158,Z 696.974,A -85,B 0,C 180,E1 -25717.338,E2 -25717.338} C_VEL
LIN {X 0,Y 157.12,Z 700.238,A -85,B 0,C 180,E1 -25719.935,E2 -25719.935} C_VEL
LIN {X 0,Y 148.833,Z 703.034,A -85,B 0,C 180,E1 -25723.542,E2 -25723.542} C_VEL
LIN {X 0,Y 141.799,Z 704.328,A -85,B 0,C 180,E1 -25727.188,E2 -25727.188} C_VEL
LIN {X 0,Y 135.035,Z 704.64,A -85,B 0,C 180,E1 -25731.433,E2 -25731.433} C_VEL
LIN {X 0,Y 128.257,Z 703.403,A -85,B 0,C 180,E1 -25736.86,E2 -25736.86} C_VEL
LIN {X 0,Y 125.133,Z 702.086,A -85,B 0,C 180,E1 -25740.001,E2 -25740.001} C_VEL
LIN {X 0,Y 121.247,Z 699.309,A -85,B 0,C 180,E1 -25744.83,E2 -25744.83} C_VEL
LIN {X 0,Y 118.112,Z 695.146,A -85,B 0,C 180,E1 -25750.284,E2 -25750.284} C_VEL
LIN {X 0,Y 116.013,Z 689.542,A -85,B 0,C 180,E1 -25756.113,E2 -25756.113} C_VEL
LIN {X 0,Y 115.085,Z 683.124,A -85,B 0,C 180,E1 -25761.496,E2 -25761.496} C_VEL
LIN {X 0,Y 115.115,Z 674.642,A -85,B 0,C 180,E1 -25767.253,E2 -25767.253} C_VEL
LIN {X 0,Y 115.88,Z 665.37,A -85,B 0,C 180,E1 -25772.257,E2 -25772.257} C_VEL
LIN {X 0,Y 117.121,Z 654.693,A -85,B 0,C 180,E1 -25776.876,E2 -25776.876} C_VEL
LIN {X 0,Y 118.573,Z 643.471,A -85,B 0,C 180,E1 -25780.693,E2 -25780.693} C_VEL
LIN {X 0,Y 120.174,Z 631.018,A -85,B 0,C 180,E1 -25783.987,E2 -25783.987} C_VEL
LIN {X 0,Y 121.525,Z 618.643,A -85,B 0,C 180,E1 -25786.467,E2 -25786.467} C_VEL
LIN {X 0,Y 122.602,Z 605.32,A -85,B 0,C 180,E1 -25788.358,E2 -25788.358} C_VEL
LIN {X 0,Y 123.33,Z 590.138,A -85,B 0,C 180,E1 -25789.829,E2 -25789.829} C_VEL
LIN {X 0,Y 115.155,Z 561.803,A -85,B 0,C 180,E1 -25793.336,E2 -25793.336} C_VEL
LIN {X 0,Y 114.976,Z 561.055,A -85,B 0,C 180,E1 -25793.962,E2 -25793.962} C_VEL
LIN {X 0,Y 114.875,Z 560.988,A -85,B 0,C 180,E1 -25800.698,E2 -25800.698} C_VEL
LIN {X 0,Y 114.95,Z 560.975,A -85,B 0,C 180,E1 -25806.509,E2 -25806.509} C_VEL
LIN {X 0,Y 115.011,Z 560.966,A -85,B 0,C 180,E1 -25812.21,E2 -25812.21} C_VEL
LIN {X 0,Y 115.258,Z 560.94,A -85,B 0,C 180,E1 -25817.328,E2 -25817.328} C_VEL
LIN {X 0,Y 115.366,Z 560.919,A -85,B 0,C 180,E1 -25823.002,E2 -25823.002} C_VEL
LIN {X 0,Y 115.996,Z 560.843,A -85,B 0,C 180,E1 -25830,E2 -25830} C_VEL
LIN {X 0,Y 115.367,Z 560.926,A -85,B 0,C 180,E1 -25836.998,E2 -25836.998} C_VEL
LIN {X 0,Y 115.253,Z 560.939,A -85,B 0,C 180,E1 -25842.659,E2 -25842.659} C_VEL
LIN {X 0,Y 115.014,Z 560.965,A -85,B 0,C 180,E1 -25847.79,E2 -25847.79} C_VEL
LIN {X 0,Y 114.95,Z 560.979,A -85,B 0,C 180,E1 -25853.491,E2 -25853.491} C_VEL
LIN {X 0,Y 114.866,Z 560.988,A -85,B 0,C 180,E1 -25861.063,E2 -25861.063} C_VEL
LIN {X 0,Y 114.849,Z 560.984,A -85,B 0,C 180,E1 -25867.729,E2 -25867.729} C_VEL
LIN {X 0,Y 114.843,Z 560.991,A -85,B 0,C 180,E1 -25872.745,E2 -25872.745} C_VEL
LIN {X 0,Y 114.837,Z 560.989,A -85,B 0,C 180,E1 -25877.684,E2 -25877.684} C_VEL
LIN {X 0,Y 114.82,Z 560.991,A -85,B 0,C 180,E1 -25882.721,E2 -25882.721} C_VEL
LIN {X 0,Y 114.869,Z 560.988,A -85,B 0,C 180,E1 -25888.931,E2 -25888.931} C_VEL
LIN {X 0,Y 114.949,Z 560.978,A -85,B 0,C 180,E1 -25896.503,E2 -25896.503} C_VEL
LIN {X 0,Y 115.02,Z 560.963,A -85,B 0,C 180,E1 -25902.21,E2 -25902.21} C_VEL
LIN {X 0,Y 115.284,Z 560.937,A -85,B 0,C 180,E1 -25907.261,E2 -25907.261} C_VEL
LIN {X 0,Y 115.388,Z 560.921,A -85,B 0,C 180,E1 -25913.002,E2 -25913.002} C_VEL
LIN {X 0,Y 115.992,Z 560.842,A -85,B 0,C 180,E1 -25919.999,E2 -25919.999} C_VEL
LIN {X 0,Y 115.383,Z 560.922,A -85,B 0,C 180,E1 -25926.996,E2 -25926.996} C_VEL
LIN {X 0,Y 115.282,Z 560.938,A -85,B 0,C 180,E1 -25932.735,E2 -25932.735} C_VEL
LIN {X 0,Y 115.01,Z 560.964,A -85,B 0,C 180,E1 -25937.789,E2 -25937.789} C_VEL
LIN {X 0,Y 114.943,Z 560.979,A -85,B 0,C 180,E1 -25943.49,E2 -25943.49} C_VEL
LIN {X 0,Y 114.86,Z 560.99,A -85,B 0,C 180,E1 -25951.062,E2 -25951.062} C_VEL
LIN {X 0,Y 114.777,Z 560.997,A -85,B 0,C 180,E1 -25957.756,E2 -25957.756} C_VEL
LIN {X 0,Y 114.785,Z 560.998,A -85,B 0,C 180,E1 -25962.717,E2 -25962.717} C_VEL
LIN {X 0,Y 114.857,Z 560.99,A -85,B 0,C 180,E1 -25967.695,E2 -25967.695} C_VEL
LIN {X 0,Y 115.805,Z 561.106,A -85,B 0,C 180,E1 -25975.991,E2 -25975.991} C_VEL
LIN {X 0,Y 116.16,Z 562.153,A -85,B 0,C 180,E1 -25976.504,E2 -25976.504} C_VEL
LIN {X 0,Y 117.416,Z 566.356,A -85,B 0,C 180,E1 -25977.102,E2 -25977.102} C_VEL
LIN {X 0,Y 117.52,Z 570.67,A -85,B 0,C 180,E1 -25977.565,E2 -25977.565} C_VEL
LIN {X 0,Y 117.4,Z 601.783,A -85,B 0,C 180,E1 -25980.835,E2 -25980.835} C_VEL
LIN {X 0,Y 119.081,Z 645.795,A -85,B 0,C 180,E1 -25985.657,E2 -25985.657} C_VEL
LIN {X 0,Y 119.597,Z 656.548,A -85,B 0,C 180,E1 -25987.317,E2 -25987.317} C_VEL
LIN {X 0,Y 118.819,Z 667.902,A -85,B 0,C 180,E1 -25989.666,E2 -25989.666} C_VEL
LIN {X 0,Y 117.809,Z 678.845,A -85,B 0,C 180,E1 -25992.646,E2 -25992.646} C_VEL
LIN {X 0,Y 116.775,Z 689.674,A -85,B 0,C 180,E1 -25996.514,E2 -25996.514} C_VEL
LIN {X 0,Y 116.424,Z 698.368,A -85,B 0,C 180,E1 -26000.444,E2 -26000.444} C_VEL
LIN {X 0,Y 116.579,Z 706.055,A -85,B 0,C 180,E1 -26004.812,E2 -26004.812} C_VEL
LIN {X 0,Y 117.339,Z 712.217,A -85,B 0,C 180,E1 -26009.142,E2 -26009.142} C_VEL
LIN {X 0,Y 117.855,Z 715.187,A -85,B 0,C 180,E1 -26011.708,E2 -26011.708} C_VEL
LIN {X 0,Y 116.178,Z 718.899,A -85,B 0,C 180,E1 -26016.949,E2 -26016.949} C_VEL
LIN {X 0,Y 115.516,Z 721.881,A -85,B 0,C 180,E1 -26023.24,E2 -26023.24} C_VEL
LIN {X 0,Y 116.057,Z 723.227,A -85,B 0,C 180,E1 -26027.624,E2 -26027.624} C_VEL
LIN {X 0,Y 118.932,Z 724.269,A -85,B 0,C 180,E1 -26034.433,E2 -26034.433} C_VEL
LIN {X 0,Y 121.187,Z 724.269,A -85,B 0,C 180,E1 -26037.641,E2 -26037.641} C_VEL
LIN {X 0,Y 127.215,Z 723.174,A -85,B 0,C 180,E1 -26043.534,E2 -26043.534} C_VEL
LIN {X 0,Y 131.193,Z 721.949,A -85,B 0,C 180,E1 -26046.531,E2 -26046.531} C_VEL
LIN {X 0,Y 139.178,Z 718.802,A -85,B 0,C 180,E1 -26051.029,E2 -26051.029} C_VEL
LIN {X 0,Y 146.323,Z 715.299,A -85,B 0,C 180,E1 -26054.141,E2 -26054.141} C_VEL
LIN {X 0,Y 156.259,Z 709.404,A -85,B 0,C 180,E1 -26057.574,E2 -26057.574} C_VEL
LIN {X 0,Y 166.518,Z 702.011,A -85,B 0,C 180,E1 -26060.375,E2 -26060.375} C_VEL
LIN {X 0,Y 175.446,Z 694.492,A -85,B 0,C 180,E1 -26062.291,E2 -26062.291} C_VEL
LIN {X 0,Y 183.216,Z 686.868,A -85,B 0,C 180,E1 -26063.66,E2 -26063.66} C_VEL
LIN {X 0,Y 192.789,Z 675.838,A -85,B 0,C 180,E1 -26065.105,E2 -26065.105} C_VEL
LIN {X 0,Y 200.772,Z 664.529,A -85,B 0,C 180,E1 -26066.416,E2 -26066.416} C_VEL
LIN {X 0,Y 201.957,Z 662.649,A -85,B 0,C 180,E1 -26066.633,E2 -26066.633} C_VEL
LIN {X 0,Y 201.93,Z 662.455,A -85,B 0,C 180,E1 -26067.163,E2 -26067.163} C_VEL
LIN {X 0,Y 200.994,Z 663.769,A -85,B 0,C 180,E1 -26067.527,E2 -26067.527} C_VEL
LIN {X 0,Y 194.38,Z 672.385,A -85,B 0,C 180,E1 -26068.988,E2 -26068.988} C_VEL
LIN {X 0,Y 188.533,Z 678.737,A -85,B 0,C 180,E1 -26070.372,E2 -26070.372} C_VEL
LIN {X 0,Y 185.865,Z 681.402,A -85,B 0,C 180,E1 -26070.795,E2 -26070.795} C_VEL
LIN {X 0,Y 176.154,Z 689.757,A -85,B 0,C 180,E1 -26071.206,E2 -26071.206} C_VEL
LIN {X 0,Y 173.133,Z 691.924,A -85,B 0,C 180,E1 -26071.667,E2 -26071.667} C_VEL
LIN {X 0,Y 172.667,Z 692.227,A -85,B 0,C 180,E1 -26071.786,E2 -26071.786} C_VEL
LIN {X 0,Y 163.227,Z 697.792,A -85,B 0,C 180,E1 -26074.497,E2 -26074.497} C_VEL
LIN {X 0,Y 154.761,Z 701.598,A -85,B 0,C 180,E1 -26077.295,E2 -26077.295} C_VEL
LIN {X 0,Y 146.79,Z 704.138,A -85,B 0,C 180,E1 -26080.42,E2 -26080.42} C_VEL
LIN {X 0,Y 138.836,Z 705.663,A -85,B 0,C 180,E1 -26084.105,E2 -26084.105} C_VEL
LIN {X 0,Y 132.371,Z 706.003,A -85,B 0,C 180,E1 -26087.74,E2 -26087.74} C_VEL
LIN {X 0,Y 128.121,Z 705.704,A -85,B 0,C 180,E1 -26090.529,E2 -26090.529} C_VEL
LIN {X 0,Y 124.199,Z 704.907,A -85,B 0,C 180,E1 -26093.503,E2 -26093.503} C_VEL
LIN {X 0,Y 119.569,Z 703.17,A -85,B 0,C 180,E1 -26097.704,E2 -26097.704} C_VEL
LIN {X 0,Y 114.684,Z 699.744,A -85,B 0,C 180,E1 -26103.515,E2 -26103.515} C_VEL
LIN {X 0,Y 111.386,Z 695.503,A -85,B 0,C 180,E1 -26109.077,E2 -26109.077} C_VEL
LIN {X 0,Y 108.95,Z 688.984,A -85,B 0,C 180,E1 -26115.816,E2 -26115.816} C_VEL
LIN {X 0,Y 107.965,Z 681.584,A -85,B 0,C 180,E1 -26121.982,E2 -26121.982} C_VEL
LIN {X 0,Y 108.13,Z 672.445,A -85,B 0,C 180,E1 -26128.115,E2 -26128.115} C_VEL
LIN {X 0,Y 108.942,Z 663.397,A -85,B 0,C 180,E1 -26133.005,E2 -26133.005} C_VEL
LIN {X 0,Y 110.329,Z 652.157,A -85,B 0,C 180,E1 -26137.817,E2 -26137.817} C_VEL
LIN {X 0,Y 111.878,Z 640.287,A -85,B 0,C 180,E1 -26141.763,E2 -26141.763} C_VEL
LIN {X 0,Y 113.4,Z 628.38,A -85,B 0,C 180,E1 -26144.829,E2 -26144.829} C_VEL
LIN {X 0,Y 114.745,Z 615.479,A -85,B 0,C 180,E1 -26147.308,E2 -26147.308} C_VEL
LIN {X 0,Y 115.816,Z 602.219,A -85,B 0,C 180,E1 -26149.08,E2 -26149.08} C_VEL
LIN {X 0,Y 116.323,Z 591.386,A -85,B 0,C 180,E1 -26150.17,E2 -26150.17} C_VEL
LIN {X 0,Y 108.094,Z 562.692,A -85,B 0,C 180,E1 -26153.932,E2 -26153.932} C_VEL
LIN {X 0,Y 107.908,Z 561.921,A -85,B 0,C 180,E1 -26154.652,E2 -26154.652} C_VEL
LIN {X 0,Y 107.816,Z 561.868,A -85,B 0,C 180,E1 -26158.569,E2 -26158.569} C_VEL
LIN {X 0,Y 107.913,Z 561.852,A -85,B 0,C 180,E1 -26166.999,E2 -26166.999} C_VEL
LIN {X 0,Y 108.031,Z 561.835,A -85,B 0,C 180,E1 -26174.918,E2 -26174.918} C_VEL
LIN {X 0,Y 108.258,Z 561.812,A -85,B 0,C 180,E1 -26178.77,E2 -26178.77} C_VEL
LIN {X 0,Y 108.447,Z 561.789,A -85,B 0,C 180,E1 -26186.285,E2 -26186.285} C_VEL
LIN {X 0,Y 108.946,Z 561.721,A -85,B 0,C 180,E1 -26190,E2 -26190} C_VEL
LIN {X 0,Y 108.306,Z 561.806,A -85,B 0,C 180,E1 -26197.457,E2 -26197.457} C_VEL
LIN {X 0,Y 108.174,Z 561.821,A -85,B 0,C 180,E1 -26202.95,E2 -26202.95} C_VEL
LIN {X 0,Y 107.907,Z 561.848,A -85,B 0,C 180,E1 -26209.005,E2 -26209.005} C_VEL
LIN {X 0,Y 107.859,Z 561.862,A -85,B 0,C 180,E1 -26214.181,E2 -26214.181} C_VEL
LIN {X 0,Y 107.798,Z 561.87,A -85,B 0,C 180,E1 -26222.051,E2 -26222.051} C_VEL
LIN {X 0,Y 107.752,Z 561.871,A -85,B 0,C 180,E1 -26228.491,E2 -26228.491} C_VEL
LIN {X 0,Y 107.719,Z 561.872,A -85,B 0,C 180,E1 -26235.862,E2 -26235.862} C_VEL
LIN {X 0,Y 107.722,Z 561.879,A -85,B 0,C 180,E1 -26241.526,E2 -26241.526} C_VEL
LIN {X 0,Y 107.807,Z 561.869,A -85,B 0,C 180,E1 -26248.564,E2 -26248.564} C_VEL
LIN {X 0,Y 107.914,Z 561.855,A -85,B 0,C 180,E1 -26256.997,E2 -26256.997} C_VEL
LIN {X 0,Y 108.039,Z 561.838,A -85,B 0,C 180,E1 -26264.917,E2 -26264.917} C_VEL
LIN {X 0,Y 108.288,Z 561.806,A -85,B 0,C 180,E1 -26268.771,E2 -26268.771} C_VEL
LIN {X 0,Y 108.456,Z 561.789,A -85,B 0,C 180,E1 -26276.283,E2 -26276.283} C_VEL
LIN {X 0,Y 108.942,Z 561.72,A -85,B 0,C 180,E1 -26279.999,E2 -26279.999} C_VEL
LIN {X 0,Y 108.324,Z 561.8,A -85,B 0,C 180,E1 -26287.454,E2 -26287.454} C_VEL
LIN {X 0,Y 108.197,Z 561.82,A -85,B 0,C 180,E1 -26293.013,E2 -26293.013} C_VEL
LIN {X 0,Y 107.902,Z 561.85,A -85,B 0,C 180,E1 -26299.005,E2 -26299.005} C_VEL
LIN {X 0,Y 107.856,Z 561.862,A -85,B 0,C 180,E1 -26304.183,E2 -26304.183} C_VEL
LIN {X 0,Y 107.782,Z 561.871,A -85,B 0,C 180,E1 -26312.042,E2 -26312.042} C_VEL
LIN {X 0,Y 107.686,Z 561.881,A -85,B 0,C 180,E1 -26318.45,E2 -26318.45} C_VEL
LIN {X 0,Y 107.709,Z 561.88,A -85,B 0,C 180,E1 -26325.867,E2 -26325.867} C_VEL
LIN {X 0,Y 108.602,Z 561.963,A -85,B 0,C 180,E1 -26335.259,E2 -26335.259} C_VEL
LIN {X 0,Y 108.968,Z 563.133,A -85,B 0,C 180,E1 -26335.871,E2 -26335.871} C_VEL
LIN {X 0,Y 110.61,Z 568.147,A -85,B 0,C 180,E1 -26336.634,E2 -26336.634} C_VEL
LIN {X 0,Y 110.343,Z 601.7,A -85,B 0,C 180,E1 -26340.39,E2 -26340.39} C_VEL
LIN {X 0,Y 111.971,Z 644.89,A -85,B 0,C 180,E1 -26345.429,E2 -26345.429} C_VEL
LIN {X 0,Y 112.449,Z 657.159,A -85,B 0,C 180,E1 -26347.493,E2 -26347.493} C_VEL
LIN {X 0,Y 111.658,Z 668.928,A -85,B 0,C 180,E1 -26350.228,E2 -26350.228} C_VEL
LIN {X 0,Y 110.663,Z 679.313,A -85,B 0,C 180,E1 -26353.421,E2 -26353.421} C_VEL
LIN {X 0,Y 109.771,Z 689.688,A -85,B 0,C 180,E1 -26357.521,E2 -26357.521} C_VEL
LIN {X 0,Y 109.568,Z 698.074,A -85,B 0,C 180,E1 -26361.702,E2 -26361.702} C_VEL
LIN {X 0,Y 109.888,Z 705.585,A -85,B 0,C 180,E1 -26366.333,E2 -26366.333} C_VEL
LIN {X 0,Y 110.902,Z 711.585,A -85,B 0,C 180,E1 -26370.907,E2 -26370.907} C_VEL
LIN {X 0,Y 111.067,Z 712.578,A -85,B 0,C 180,E1 -26371.813,E2 -26371.813} C_VEL
LIN {X 0,Y 109.941,Z 715.439,A -85,B 0,C 180,E1 -26375.502,E2 -26375.502} C_VEL
LIN {X 0,Y 108.889,Z 718.587,A -85,B 0,C 180,E1 -26381.164,E2 -26381.164} C_VEL
LIN {X 0,Y 109.489,Z 721.379,A -85,B 0,C 180,E1 -26388.719,E2 -26388.719} C_VEL
